# B&R Automation Studio project NAINV104C00R8L515F00 (part 10)

#### Act_OptC0011Loading.st
```iecst
ACTION Act_OptC0011Loading:
	fbLoadingWarmUpTm.PT := p_tyNtParamCurr.tComLoadRstTm ;
	udiElapseTm := (TIME_TO_UDINT (fbLoadingWarmUpTm.PT )- TIME_TO_UDINT (fbLoadingWarmUpTm.ET))/1000;
	sElapseTm := UDINT_TO_STRING(udiElapseTm);

	//Loading When Reset pressed
	IF bLoadingScreen=TRUE THEN

		fUIInRtStatOff(ADR(tyCommon.tyLoading.tyLyr.uiRtStat));
	ELSE
		fUIInRtStatHide(ADR(tyCommon.tyLoading.tyLyr.uiRtStat));
	END_IF

	IF fbLoadingWarmUpTm.Q = FALSE THEN
		tyCommon.tyLoading.tyStringMsg.sValue := CONCAT('Please wait for ',sElapseTm);
		tyCommon.tyLoading.tyStringMsg.sValue := CONCAT(tyCommon.tyLoading.tyStringMsg.sValue,' seconds...');
	END_IF

	fbLoadingWarmUpTm (IN := TRUE);
	fbLoadingLogoTm	(IN := TRUE);

	// ADD
	IF fbLoadingWarmUpTm.Q = FALSE  AND tyCommon.tyLoading.tyLyr.uiRtStat = 0 THEN
		IF fbLoadingLogoTm.Q = TRUE AND tyCommon.tyLoading.tyUILoad.usiValueIdx <= 2 THEN
			tyCommon.tyLoading.tyUILoad.usiValueIdx := (tyCommon.tyLoading.tyUILoad.usiValueIdx) +1 ;
			fbLoadingLogoTm (IN := FALSE);
			fbLoadingLogoTm (IN := TRUE);
		ELSIF fbLoadingLogoTm.Q = TRUE AND tyCommon.tyLoading.tyUILoad.usiValueIdx > 2 THEN
			tyCommon.tyLoading.tyUILoad.usiValueIdx := 0;
			fbLoadingLogoTm (IN := FALSE);
			fbLoadingLogoTm (IN := TRUE);
		END_IF
	ELSE	// fbLoadingWarmUpTm.Q = TRUE
		//fUIInRtStatHide(ADR(tyCommon.tyLoading.tyLyr.uiRtStat));
		bLoadingScreen:= FALSE;
		fbLoadingWarmUpTm (IN := FALSE);
		fbLoadingLogoTm (IN := FALSE);
	END_IF

END_ACTION
```

#### Act_EntP0000Disp.st
```iecst
ACTION Act_EntP0000Disp:

	//Access Address
	p_tyP0000SSaver ACCESS ADR(tyP0000SSaver.tySSaver);

END_ACTION
```

#### Act_OptP0000McStatus.st
```iecst
ACTION Act_OptP0000McStatus:

	IF p_bAlarmErr = TRUE THEN
		tyP0000SSaver.tySSaver.tyTxtMcStat.usiValueIdx	:= 6;

	ELSIF p_bAlarmWarning = TRUE THEN
		tyP0000SSaver.tySSaver.tyTxtMcStat.usiValueIdx	:= 7;

	ELSIF p_eOpsOpsStatus = OperationsStatusRun THEN

		tyP0000SSaver.tySSaver.tyTxtMcStat.usiValueIdx	:= 1;

//	ELSIF tyOpsProgData.bSimuCtrl = TRUE THEN
//		tyP0000SSaver.tySSaver.tyTxtMcStat.usiValueIdx	:= 5;

	ELSIF bUIManualMod = TRUE THEN
		tyP0000SSaver.tySSaver.tyTxtMcStat.usiValueIdx	:= 3;

	ELSE
		tyP0000SSaver.tySSaver.tyTxtMcStat.usiValueIdx	:= 2;

	END_IF

END_ACTION
```

#### Act_OptP0000RunningNm.st
```iecst
ACTION Act_OptP0000RunningNm:
	fbSSaverTm(IN := TRUE , PT := T#2s);

	IF EDGEPOS(fbSSaverTm.Q = FALSE) THEN
		CASE uiSSaverCnt OF
			0:
				tyP0000SSaver.tySSaver.tyTxtMcNm.sValue	:= CONCAT(p_tyMcParamCurr.sMcNm , '                                        ');
			1:
				tyP0000SSaver.tySSaver.tyTxtMcNm.sValue	:= CONCAT('          ' , CONCAT(p_tyMcParamCurr.sMcNm , '                              '));
			2:
				tyP0000SSaver.tySSaver.tyTxtMcNm.sValue	:= CONCAT('                    ' , CONCAT(p_tyMcParamCurr.sMcNm , '                    '));
			3:
				tyP0000SSaver.tySSaver.tyTxtMcNm.sValue	:= CONCAT('                              ' , CONCAT(p_tyMcParamCurr.sMcNm , '          '));
			4:
				tyP0000SSaver.tySSaver.tyTxtMcNm.sValue	:= CONCAT('                                        ' , p_tyMcParamCurr.sMcNm);
			5:
				tyP0000SSaver.tySSaver.tyTxtMcNm.sValue	:= CONCAT('                              ' , CONCAT(p_tyMcParamCurr.sMcNm , '          '));
			6:
				tyP0000SSaver.tySSaver.tyTxtMcNm.sValue	:= CONCAT('                    ' , CONCAT(p_tyMcParamCurr.sMcNm , '                    '));
			7:
				tyP0000SSaver.tySSaver.tyTxtMcNm.sValue	:= CONCAT('          ' , CONCAT(p_tyMcParamCurr.sMcNm , '                              '));

		END_CASE

	END_IF

	IF fbSSaverTm.Q = TRUE THEN
		fbSSaverTm(IN := FALSE);
		uiSSaverCnt	:= uiSSaverCnt + 1;
		IF uiSSaverCnt = 8 THEN
			uiSSaverCnt	:= 0;
		END_IF
	END_IF

END_ACTION
```

#### Act_OptP0000DisableSSaver.st
```iecst
ACTION Act_OptP0000DisableSSaver:

	IF p_tyNtParamCurr.bSSaverPrep = FALSE OR p_tyMcParamCurr.bSSaverEn = FALSE THEN

		IF tyProperty.tyVisu.uiSSaverRemainTm < 5 THEN
			tyProperty.tyVisu.uiSSaverTm	:= 9;
		ELSE
			tyProperty.tyVisu.uiSSaverTm	:= 10;
		END_IF

	END_IF

	IF EDGEPOS(p_tyNtParamCurr.bSSaverPrep AND p_tyMcParamCurr.bSSaverEn) THEN
		tyProperty.tyVisu.uiSSaverTm	:= p_tyMcParamCurr.uiSSaverTmInSec;
	END_IF

END_ACTION
```

#### Act_OptP0000StatDisp.st
```iecst
ACTION Act_OptP0000StatDisp:

	//Error / Warning / Info
	IF p_bAlarmErr = TRUE OR p_bAlarmWarning = TRUE OR p_bAlarmInfo = TRUE THEN

		fbErrBlinkTm(IN := TRUE);
		IF fbErrBlinkTm.Q = TRUE THEN
			fbErrBlinkTm(IN := FALSE);

			IF p_bAlarmErr THEN

				IF tyP0000SSaver.tySSaver.tyBitmapStat.usiValueIdx = 1 THEN
					tyP0000SSaver.tySSaver.tyBitmapStat.usiValueIdx	:= 0;
				ELSE
					tyP0000SSaver.tySSaver.tyBitmapStat.usiValueIdx	:= 1;
				END_IF

			ELSE

				IF tyP0000SSaver.tySSaver.tyBitmapStat.usiValueIdx = 3 THEN
					tyP0000SSaver.tySSaver.tyBitmapStat.usiValueIdx	:= 0;
				ELSE
					tyP0000SSaver.tySSaver.tyBitmapStat.usiValueIdx	:= 3;
				END_IF

			END_IF

		END_IF

	//Safety Relay Signal Activated
	ELSIF p_tyDI.bSafetyRlySig = FALSE THEN

		fbRstBlinkTm(IN := TRUE);
		IF fbRstBlinkTm.Q = TRUE THEN
			fbRstBlinkTm(IN := FALSE);

			IF tyP0000SSaver.tySSaver.tyBitmapStat.usiValueIdx = 5 THEN
				tyP0000SSaver.tySSaver.tyBitmapStat.usiValueIdx			:= 6;
			ELSE
				tyP0000SSaver.tySSaver.tyBitmapStat.usiValueIdx			:= 5;
			END_IF

		END_IF

	//Manual Running
	ELSIF bUIManualMod THEN
		tyP0000SSaver.tySSaver.tyBitmapStat.usiValueIdx	:= 7;

	//Operation Cycle Stopping
	ELSIF p_eOpsOpsStatus = OperationsStatusCycleStopping THEN

		fbStopBlinkTm(IN := TRUE);
		IF fbStopBlinkTm.Q = TRUE THEN
			fbStopBlinkTm(IN := FALSE);

			IF tyP0000SSaver.tySSaver.tyBitmapStat.usiValueIdx = 1 THEN
				tyP0000SSaver.tySSaver.tyBitmapStat.usiValueIdx	:= 2;
			ELSE
				tyP0000SSaver.tySSaver.tyBitmapStat.usiValueIdx	:= 1;
			END_IF

		END_IF

	//Operation Stepping
	ELSIF p_eOpsOpsStatus = OperationsStatusStep THEN
		tyP0000SSaver.tySSaver.tyBitmapStat.usiValueIdx	:= 3;

	//Operation Running
	ELSIF p_eOpsOpsStatus = OperationsStatusRun THEN
		tyP0000SSaver.tySSaver.tyBitmapStat.usiValueIdx	:= 2;

	//Standby
	ELSE
		tyP0000SSaver.tySSaver.tyBitmapStat.usiValueIdx	:= 0;

	END_IF

END_ACTION
```

#### Act_OptP0000TouchTimer.st
```iecst
ACTION Act_OptP0000TouchTimer:

	IF bLoginSuccess AND p_tyNtParamCurr.bAutoLogoutPrep AND p_tyMcParamCurr.bAutoLogoutEn THEN

		fbTouchTm();

		fbAutoLogoutTm(IN:= NOT fbTouchTm.bPressed, PT:=DINT_TO_TIME(p_tyMcParamCurr.diAutoLogoutTmInSec));

		//Reset Time When Pressed
		IF fbTouchTm.bPressed THEN
			fbAutoLogoutTm(IN:=FALSE);
		END_IF

		//Auto Logout
		IF fbAutoLogoutTm.Q THEN

			bPromptSessionExp	:= TRUE;
			p_tyC0008MsgBox ACCESS ADR(tyP0000SSaver.tyMsgBoxLoginAsk);

			IF bChgPageDone=FALSE THEN

				IF eCurrPage<>UIP0002Menu THEN
					CASE eCurrPage OF

						UIP0900GenIn, UIP0910GenOut, UIP0920MtrNPneuCtrl, UIP0923Stopper, UIP0931ConvInv, UIP0934AW, UIP0940CommCtrl:

							eChgPage		:= UIP0002Menu;

							tyP0002Menu.tyMenu.tyBtnMnlRst.bRtCompl := TRUE ;

							bChgPageDone	:= TRUE;

						UIP1000Lang, UIP1021McSetGen, UIP1022McSetVComm, UIP1023McSetHComm, UIP1024McSetAntiGap:

							IF tyCommon.tySet.tyBtnSave.uiMaskRtStat.0 = FALSE THEN

								eChgPage	:= UIP0002Menu;

								bChgPageDone	:= TRUE;

							ELSE

								eChgPage		:= UIP0002Menu;

								IF eCurrPage= UIP1021McSetGen THEN

									tyP1021McSetGen.tyMsgBoxExitAsk.tyBtnYes.bRtCompl := TRUE;

									bChgPageDone	:= TRUE;

								ELSIF eCurrPage= UIP1022McSetVComm THEN

									tyP1022McSetVComm.tyMsgBoxExitAsk.tyBtnYes.bRtCompl := TRUE;

									bChgPageDone	:= TRUE;

								ELSIF eCurrPage= UIP1023McSetHComm THEN

									tyP1023McSetHComm.tyMsgBoxExitAsk.tyBtnYes.bRtCompl := TRUE;

									bChgPageDone	:= TRUE;

								ELSIF eCurrPage= UIP1024McSetAntiGap THEN

									tyP1024McSetAntiGap.tyMsgBoxExitAsk.tyBtnYes.bRtCompl := TRUE;

									bChgPageDone	:= TRUE;

								ELSE  //language page
									bChgPageDone	:= TRUE;
								END_IF

							END_IF

						ELSE
							eChgPage		:= UIP0002Menu;

							bChgPageDone	:= TRUE;

					END_CASE

				ELSE
					bChgPageDone	:= TRUE;
				END_IF

			END_IF

			IF bChgPageDone THEN

				eUsrMgmtAct	:= UsrMgmtActLogout;

				IF p_eUsrMgmtStat = UsrMgmtActLogout AND p_eUsrMgmtStatus = Done THEN
					eUsrMgmtAct	:= UsrMgmtActIdle;

					bLoginSuccess	:= FALSE;

					bChgPageDone	:= FALSE;

					fbAutoLogoutTm(IN:=FALSE);

				END_IF

			END_IF

		END_IF

	ELSE
		fbAutoLogoutTm(IN:=FALSE);
		bChgPageDone	:= FALSE;
	END_IF

	//Prompt Relogin After Auto Logout
	IF tyP0000SSaver.tyMsgBoxLoginAsk.tyBtnYes.bRtCompl = TRUE THEN
		tyP0000SSaver.tyMsgBoxLoginAsk.tyBtnYes.bRtCompl 	:= FALSE;
		tyP0000SSaver.tyMsgBoxLoginAsk.tyBtnYes.bValue		:= FALSE;
		p_tyC0008MsgBox ACCESS ADR(tyP0000SSaver.tyMsgBoxHide);
		bPromptSessionExp	:= FALSE;

	ELSIF tyP0000SSaver.tyMsgBoxLoginAsk.tyBtnNo.bRtCompl = TRUE THEN
		tyP0000SSaver.tyMsgBoxLoginAsk.tyBtnNo.bRtCompl 	:= FALSE;
		tyP0000SSaver.tyMsgBoxLoginAsk.tyBtnNo.bValue		:= FALSE;
		p_tyC0008MsgBox ACCESS ADR(tyP0000SSaver.tyMsgBoxHide);
		eChgPage		:= UIP0100Login;
		bPromptSessionExp	:= FALSE;

	END_IF

END_ACTION
```

#### Act_EntP0001Disp.st
```iecst
ACTION Act_EntP0001Disp:

	//UI Property Access Address
	p_tyVisu ACCESS ADR(tyProperty.tyVisu);

	p_tyKeypad ACCESS ADR(tyProperty.tyKeypad);

	p_tyTxtSnippets ACCESS ADR(tyProperty.tyUITxtSnippets);

	p_tyC0008MsgBox ACCESS ADR(tyP0001Startup.tyMsgBoxHide);

	//Access Address
	p_tyP0001Startup ACCESS ADR(tyP0001Startup.tyStartup);

	p_tyP0001Initial ACCESS ADR(tyP0001Startup.tyInitial);

	fUIInRtStatHide(ADR(tyP0001Startup.tyInitial.tyLyr.uiRtStat));

END_ACTION
```

#### Act_OptP0001Startup.st
```iecst
ACTION Act_OptP0001Startup:

	//Screen Saver
	p_tyP0000SSaver ACCESS ADR(tyP0000SSaver.tySSaver);

	IF (eChgPage = UIP0001Startup) OR (eCurrPage = UIP0001Startup) THEN

		eStartupAct		:= StartupActRun;

		IF p_eStartupStat = StartupActRun AND p_eStartupStatus = Done THEN
			eStartupAct	:= StartupActIdle;

			IF p_bAlarmErr OR p_bAlarmWarning THEN
				eChgPage	:= UIP0600Alm;
			ELSE
				eChgPage	:= UIP0002Menu;
			END_IF

		END_IF

	END_IF

	tyP0001Startup.tyStartup.tyBarGraphStartup.iValue	:= DINT_TO_INT(p_eStartupStep + 1);
	tyP0001Startup.tyStartup.tyTxtStartupStat.sTxt		:= p_sStartupStepTxt;

	//IP Config
	IF DiagCpuIsSimulated() = FALSE THEN
		IF p_eStartupStep>1 THEN

			IF p_bStartupGetConfigDone THEN
				IF bTempAddrFillDone=FALSE THEN

					tyMcParamWr:= p_tyMcParamCurr;

					sTempIPAddr 	:= p_sHWInfoIPAddr;
					sTempSubnetMask	:= p_sHWInfoSubnetMask;
					udiTempEthMode	:= p_udiHWInfoEthMode;

					bTempAddrFillDone	:= TRUE;
				END_IF
			END_IF

			IF bTempAddrFillDone THEN

				IF bIPConfigChgDone=FALSE THEN

					IF  (p_tyMcParamCurr.eNetworkMod = UDINT_TO_DINT(udiTempEthMode)) AND (p_tyMcParamCurr.sIPAddr = sTempIPAddr) AND (p_tyMcParamCurr.sSubnetMask = sTempSubnetMask) THEN

						p_tyC0008MsgBox ACCESS ADR(tyP0001Startup.tyMsgBoxHide);
					ELSE
						IF p_bStartupMismatchSetConfigDone THEN

							IF (p_tyMcParamCurr.eNetworkMod <> UDINT_TO_DINT(udiTempEthMode)) THEN
								tyP0001Startup.tyMsgBoxIPConfig.tyTxtMsg.usiValueIdx := 194;
							ELSIF (p_tyMcParamCurr.sIPAddr <> sTempIPAddr) AND (p_tyMcParamCurr.sSubnetMask <> sTempSubnetMask) THEN
								tyP0001Startup.tyMsgBoxIPConfig.tyTxtMsg.usiValueIdx := 193;
							ELSIF (p_tyMcParamCurr.sIPAddr <> sTempIPAddr) THEN
								tyP0001Startup.tyMsgBoxIPConfig.tyTxtMsg.usiValueIdx := 191;
							ELSE
								tyP0001Startup.tyMsgBoxIPConfig.tyTxtMsg.usiValueIdx := 192;
							END_IF

							p_tyC0008MsgBox ACCESS ADR(tyP0001Startup.tyMsgBoxIPConfig);

						ELSE
							sSetIPAddr				:= p_tyMcParamCurr.sIPAddr;
							sSetSubnetMask			:= p_tyMcParamCurr.sSubnetMask;
							usiNetworkModeSelected	:= DINT_TO_USINT(p_tyMcParamCurr.eNetworkMod);

							bMismatchOverWriteConfig			:= TRUE;
						END_IF

					END_IF
				END_IF
			END_IF
		END_IF
	END_IF

	IF tyP0001Startup.tyMsgBoxIPConfig.tyBtnYes.bRtCompl = TRUE THEN
		tyP0001Startup.tyMsgBoxIPConfig.tyBtnYes.bRtCompl	:= FALSE;
		tyP0001Startup.tyMsgBoxIPConfig.tyBtnYes.bValue	:= FALSE;

		bIPConfigChgDone	:= TRUE;

		p_tyC0008MsgBox ACCESS ADR(tyP0001Startup.tyMsgBoxHide);

	ELSIF tyP0001Startup.tyMsgBoxIPConfig.tyBtnNo.bRtCompl = TRUE THEN

		IF (p_tyMcParamCurr.eNetworkMod <> UDINT_TO_DINT(udiTempEthMode))  THEN

			IF udiTempEthMode = DINT_TO_UDINT(IPFromDHCPServer) THEN

				bOverwriteEthMode	:= TRUE;
				bOverwriteIP 		:= FALSE;
				bOverwriteSubnet	:= FALSE;

				usiNetworkModeSelected	:= UDINT_TO_USINT(udiTempEthMode);

				tyMcParamWr.eNetworkMod	:= UDINT_TO_DINT(udiTempEthMode);

				bIPConfigChgDone	:= TRUE;

				tyP0001Startup.tyMsgBoxIPConfig.tyBtnNo.bRtCompl:= FALSE;
				tyP0001Startup.tyMsgBoxIPConfig.tyBtnNo.bValue	:= FALSE;

				p_tyC0008MsgBox ACCESS ADR(tyP0001Startup.tyMsgBoxHide);
			ELSE
				bOverwriteEthMode	:= TRUE;
				bOverwriteIP 		:= TRUE;
				bOverwriteSubnet	:= TRUE;

				usiNetworkModeSelected	:= UDINT_TO_USINT(udiTempEthMode);
				sSetIPAddr				:= sTempIPAddr;
				sSetSubnetMask			:= sTempSubnetMask;

				tyMcParamWr.eNetworkMod			:= UDINT_TO_DINT(udiTempEthMode);
				tyMcParamWr.sIPAddr				:= sTempIPAddr;
				tyMcParamWr.sSubnetMask			:= sTempSubnetMask;

				bIPConfigChgDone	:= TRUE;

				tyP0001Startup.tyMsgBoxIPConfig.tyBtnNo.bRtCompl:= FALSE;
				tyP0001Startup.tyMsgBoxIPConfig.tyBtnNo.bValue	:= FALSE;

				p_tyC0008MsgBox ACCESS ADR(tyP0001Startup.tyMsgBoxHide);
			END_IF

		ELSE

			IF (p_tyMcParamCurr.sIPAddr <> sTempIPAddr) AND (p_tyMcParamCurr.sSubnetMask <> sTempSubnetMask) THEN

				bOverwriteEthMode	:= FALSE;
				bOverwriteIP 		:= TRUE;
				bOverwriteSubnet	:= TRUE;

				sSetIPAddr		:= sTempIPAddr;
				sSetSubnetMask	:= sTempSubnetMask;

				tyMcParamWr.sIPAddr				:= sTempIPAddr;
				tyMcParamWr.sSubnetMask			:= sTempSubnetMask;

				bIPConfigChgDone	:= TRUE;

				tyP0001Startup.tyMsgBoxIPConfig.tyBtnNo.bRtCompl	:= FALSE;
				tyP0001Startup.tyMsgBoxIPConfig.tyBtnNo.bValue	:= FALSE;

				p_tyC0008MsgBox ACCESS ADR(tyP0001Startup.tyMsgBoxHide);

			ELSIF (p_tyMcParamCurr.sIPAddr <> sTempIPAddr) THEN

				bOverwriteEthMode	:= FALSE;
				bOverwriteIP 		:= TRUE;
				bOverwriteSubnet	:= FALSE;

				sSetIPAddr			:= sTempIPAddr;

				tyMcParamWr.sIPAddr	:= sTempIPAddr;

				bIPConfigChgDone	:= TRUE;

				tyP0001Startup.tyMsgBoxIPConfig.tyBtnNo.bRtCompl	:= FALSE;
				tyP0001Startup.tyMsgBoxIPConfig.tyBtnNo.bValue	:= FALSE;

				p_tyC0008MsgBox ACCESS ADR(tyP0001Startup.tyMsgBoxHide);
			ELSE

				bOverwriteEthMode	:= FALSE;
				bOverwriteIP 		:= FALSE;
				bOverwriteSubnet	:= TRUE;

				sSetSubnetMask	:= sTempSubnetMask;

				tyMcParamWr.sSubnetMask			:= sTempSubnetMask;

				bIPConfigChgDone				:= TRUE;

				tyP0001Startup.tyMsgBoxIPConfig.tyBtnNo.bRtCompl	:= FALSE;
				tyP0001Startup.tyMsgBoxIPConfig.tyBtnNo.bValue		:= FALSE;

				p_tyC0008MsgBox ACCESS ADR(tyP0001Startup.tyMsgBoxHide);
			END_IF
		END_IF
	END_IF

END_ACTION
```

#### Act_EntP0002Disp.st
```iecst
ACTION Act_EntP0002Disp:

	//Access Address
	p_tyC0005Main ACCESS ADR(tyCommon.tyMain);

	p_tyC0007Notif ACCESS ADR(tyCommon.tyNotif);

	IF NOT bPromptSessionExp THEN
		p_tyC0008MsgBox ACCESS ADR(tyP0002Menu.tyMsgBoxHide);
	END_IF

	p_tyC0009Info ACCESS ADR(tyCommon.tyInfo);

	p_tyP0002Menu ACCESS ADR(tyP0002Menu.tyMenu);

	p_tyC0011Loading ACCESS ADR(tyCommon.tyLoading);

	//Display
	//Leader Follower
	IF p_tyNtParamCurr.bLFPrep = TRUE AND p_tyMcParamCurr.bLFEn = TRUE AND ((NOT p_tyNtParamCurr.bLFUsrSetPrep AND p_tyNtParamCurr.bLeaderMc) OR (p_tyNtParamCurr.bLFUsrSetPrep AND p_tyMcParamCurr.bLFLeaderMc)) AND p_tyMcParamCurr.eUSComm <> McSetCommModHermes THEN
		fUIInRtStatOff(ADR(tyP0002Menu.tyMenu.tyBtnLFSet.uiRtStat));
		fUIInRtStatOff(ADR(tyP0002Menu.tyMenu.tyBtnLFCtrl.uiRtStat));
	ELSE
		fUIInRtStatHide(ADR(tyP0002Menu.tyMenu.tyBtnLFSet.uiRtStat));
		fUIInRtStatHide(ADR(tyP0002Menu.tyMenu.tyBtnLFCtrl.uiRtStat));
	END_IF

	//Login/Logout
	IF bLoginSuccess = FALSE THEN
		tyP0002Menu.tyMenu.tyBtnLogin.usiBitmapIdx	:= 0;
		tyP0002Menu.tyMenu.tyBtnLogin.usiTxtIdx		:= 0;
	ELSE
		tyP0002Menu.tyMenu.tyBtnLogin.usiBitmapIdx	:= 1;
		tyP0002Menu.tyMenu.tyBtnLogin.usiTxtIdx		:= 1;
	END_IF

	//Mask
	Act_OptP0002Mask;

END_ACTION
```

#### Act_OptP0002Navi.st
```iecst
ACTION Act_OptP0002Navi:

	IF (tyP0002Menu.tyMnl.tyHotspotGen.bRtCompl = TRUE) OR (tyP0002Menu.tySet.tyHotspotGen.bRtCompl = TRUE) THEN
		tyP0002Menu.tyMnl.tyHotspotGen.bRtCompl	:= FALSE;
		tyP0002Menu.tySet.tyHotspotGen.bRtCompl	:= FALSE;

		fUIInRtStatOff(ADR(tyP0002Menu.tyGen.tyLyr.uiRtStat));
		fUIInRtStatHide(ADR(tyP0002Menu.tyMnl.tyLyr.uiRtStat));
		fUIInRtStatHide(ADR(tyP0002Menu.tySet.tyLyr.uiRtStat));

	ELSIF (tyP0002Menu.tyGen.tyHotspotMnl.bRtCompl = TRUE) OR (tyP0002Menu.tySet.tyHotspotMnl.bRtCompl = TRUE) THEN
		tyP0002Menu.tyGen.tyHotspotMnl.bRtCompl	:= FALSE;
		tyP0002Menu.tySet.tyHotspotMnl.bRtCompl	:= FALSE;

		fUIInRtStatHide(ADR(tyP0002Menu.tyGen.tyLyr.uiRtStat));
		fUIInRtStatOff(ADR(tyP0002Menu.tyMnl.tyLyr.uiRtStat));
		fUIInRtStatHide(ADR(tyP0002Menu.tySet.tyLyr.uiRtStat));

	ELSIF (tyP0002Menu.tyGen.tyHotspotSet.bRtCompl = TRUE) OR (tyP0002Menu.tyMnl.tyHotspotSet.bRtCompl = TRUE) THEN
		tyP0002Menu.tyGen.tyHotspotSet.bRtCompl	:= FALSE;
		tyP0002Menu.tyMnl.tyHotspotSet.bRtCompl	:= FALSE;

		fUIInRtStatHide(ADR(tyP0002Menu.tyGen.tyLyr.uiRtStat));
		fUIInRtStatHide(ADR(tyP0002Menu.tyMnl.tyLyr.uiRtStat));
		fUIInRtStatOff(ADR(tyP0002Menu.tySet.tyLyr.uiRtStat));

	END_IF

END_ACTION
```

#### Act_OptP0002ChgPage.st
```iecst
ACTION Act_OptP0002ChgPage:

	//General
	IF tyP0002Menu.tyMenu.tyBtnOpt.bRtCompl = TRUE THEN
		tyP0002Menu.tyMenu.tyBtnOpt.bRtCompl	:= FALSE;

		eChgPage	:= UIP0200OpsGen;

	ELSIF tyP0002Menu.tyMenu.tyBtnProdSel.bRtCompl = TRUE THEN
		tyP0002Menu.tyMenu.tyBtnProdSel.bRtCompl:= FALSE;

		eChgPage	:= UIP0400ProdSel;

	ELSIF tyP0002Menu.tyMenu.tyBtnMcInfo.bRtCompl = TRUE THEN
		tyP0002Menu.tyMenu.tyBtnMcInfo.bRtCompl	:= FALSE;

		eChgPage := UIP0300McInfo;

	ELSIF tyP0002Menu.tyMenu.tyBtnAlm.bRtCompl = TRUE THEN
		tyP0002Menu.tyMenu.tyBtnAlm.bRtCompl	:= FALSE;

		eChgPage	:= UIP0600Alm;

	ELSIF tyP0002Menu.tyMenu.tyBtnLogin.bRtCompl = TRUE THEN
		tyP0002Menu.tyMenu.tyBtnLogin.bRtCompl	:= FALSE;

		eChgPage	:= UIP0100Login;

	ELSIF tyP0002Menu.tyMenu.tyBtnLFCtrl.bRtCompl = TRUE THEN
		tyP0002Menu.tyMenu.tyBtnLFCtrl.bRtCompl	:= FALSE;

		eChgPage	:= UIP0700LFCtrl;

	//Manual
	ELSIF tyP0002Menu.tyMenu.tyBtnGenInput.bRtCompl = TRUE THEN
		tyP0002Menu.tyMenu.tyBtnGenInput.bRtCompl	:= FALSE;

		bUIManualMod	:= TRUE;

		eChgPage	:= UIP0900GenIn;

	ELSIF tyP0002Menu.tyMenu.tyBtnGenOutput.bRtCompl = TRUE THEN
		tyP0002Menu.tyMenu.tyBtnGenOutput.bRtCompl	:= FALSE;

		bUIManualMod	:= TRUE;

		eChgPage	:= UIP0910GenOut;

	ELSIF tyP0002Menu.tyMenu.tyBtnMovCtrl.bRtCompl = TRUE THEN
		tyP0002Menu.tyMenu.tyBtnMovCtrl.bRtCompl	:= FALSE;

		bUIManualMod	:= TRUE;

		eChgPage	:= UIP0920MtrNPneuCtrl;

	ELSIF tyP0002Menu.tyMenu.tyBtnCommCtrl.bRtCompl = TRUE THEN
		tyP0002Menu.tyMenu.tyBtnCommCtrl.bRtCompl	:= FALSE;

		bUIManualMod	:= TRUE;

		eChgPage	:= UIP0940CommCtrl;

	ELSIF tyP0002Menu.tyMenu.tyBtnSimu.bRtCompl = TRUE THEN
		tyP0002Menu.tyMenu.tyBtnSimu.bRtCompl	:= FALSE;

		eChgPage	:= UIP0950Simu;

	//Settings
	ELSIF tyP0002Menu.tyMenu.tyBtnLang.bRtCompl = TRUE THEN
		tyP0002Menu.tyMenu.tyBtnLang.bRtCompl	:= FALSE;

		eChgPage	:= UIP1000Lang;

	ELSIF tyP0002Menu.tyMenu.tyBtnMcSet.bRtCompl = TRUE THEN
		tyP0002Menu.tyMenu.tyBtnMcSet.bRtCompl	:= FALSE;

		eChgPage	:= UIP1020McSetNavi;

	ELSIF tyP0002Menu.tyMenu.tyBtnProdSet.bRtCompl = TRUE THEN
		tyP0002Menu.tyMenu.tyBtnProdSet.bRtCompl:= FALSE;

		eChgPage	:= UIP1040ProdSet;

	ELSIF tyP0002Menu.tyMenu.tyBtnLFSet.bRtCompl = TRUE THEN
		tyP0002Menu.tyMenu.tyBtnLFSet.bRtCompl	:= FALSE;

		eChgPage	:= UIP1050LFSet;

	ELSIF tyP0002Menu.tyMenu.tyBtnUsrMgmt.bRtCompl = TRUE THEN
		tyP0002Menu.tyMenu.tyBtnUsrMgmt.bRtCompl:= FALSE;

		eChgPage	:= UIP1080UsrMgmt;

	END_IF

END_ACTION
```

#### Act_OptP0002Mask.st
```iecst
ACTION Act_OptP0002Mask:

	tyP0002Menu.tyMenu.tyBtnOpt.uiMaskRtStat.0 			:= p_tyUsrMgmtCurrAccessRgt.bOpt;
	tyP0002Menu.tyMenu.tyBtnProdSel.uiMaskRtStat.0 		:= p_tyUsrMgmtCurrAccessRgt.bProdSel AND p_bOpsStatusStop;
	tyP0002Menu.tyMenu.tyBtnMcInfo.uiMaskRtStat.0 		:= p_tyUsrMgmtCurrAccessRgt.bMcInfo;
	tyP0002Menu.tyMenu.tyBtnAlm.uiMaskRtStat.0 			:= p_tyUsrMgmtCurrAccessRgt.bAlm;
	tyP0002Menu.tyMenu.tyBtnLogin.uiMaskRtStat.0		:= p_bOpsStatusStop;
	tyP0002Menu.tyMenu.tyBtnLFCtrl.uiMaskRtStat.0 		:= p_tyUsrMgmtCurrAccessRgt.bLFCtrl;
	tyP0002Menu.tyMenu.tyBtnGenInput.uiMaskRtStat.0 	:= p_tyUsrMgmtCurrAccessRgt.bManual AND p_bOpsStatusStop;
	tyP0002Menu.tyMenu.tyBtnGenOutput.uiMaskRtStat.0 	:= p_tyUsrMgmtCurrAccessRgt.bManual AND p_bOpsStatusStop;
	tyP0002Menu.tyMenu.tyBtnMovCtrl.uiMaskRtStat.0 		:= p_tyUsrMgmtCurrAccessRgt.bManual AND p_bOpsStatusStop;
	tyP0002Menu.tyMenu.tyBtnCommCtrl.uiMaskRtStat.0 	:= p_tyUsrMgmtCurrAccessRgt.bManual AND p_bOpsStatusStop;
	tyP0002Menu.tyMenu.tyBtnSimu.uiMaskRtStat.0 		:= p_tyUsrMgmtCurrAccessRgt.bSimulation AND p_bOpsStatusStop;
	tyP0002Menu.tyMenu.tyBtnProdSet.uiMaskRtStat.0 		:= p_tyUsrMgmtCurrAccessRgt.bProdSet AND p_bOpsStatusStop;
	tyP0002Menu.tyMenu.tyBtnMcSet.uiMaskRtStat.0 		:= p_tyUsrMgmtCurrAccessRgt.bMcSet AND p_bOpsStatusStop;
	tyP0002Menu.tyMenu.tyBtnLang.uiMaskRtStat.0 		:= p_tyUsrMgmtCurrAccessRgt.bLang AND p_bOpsStatusStop;
	tyP0002Menu.tyMenu.tyBtnUsrMgmt.uiMaskRtStat.0 		:= p_tyUsrMgmtCurrAccessRgt.bUsrMgmt AND p_bOpsStatusStop;
	tyP0002Menu.tyMenu.tyBtnLFSet.uiMaskRtStat.0 		:= p_tyUsrMgmtCurrAccessRgt.bLFSet AND p_bOpsStatusStop;

	tyP0002Menu.tyMenu.tyBitmapMaskProdSetLCS.uiMaskRtStat.0	:= NOT(p_tyNtParamCurr.bLCSManageRcpPrep AND p_tyMcParamCurr.bLCSManageRcpEn);

END_ACTION
```

#### Act_OptP0002ManualCtrl.st
```iecst
ACTION Act_OptP0002ManualCtrl:

	IF EDGEPOS(bUIManualMod) THEN

		IF p_tyNtParamCurr.eTLBuzMode= TLBuzModBHTC THEN

			tyP0910GenOut.tyGenOut.tyBtnTLWhite.bValue	:= TRUE;
		ELSE

			tyP0910GenOut.tyGenOut.tyBtnTLAmber.bValue	:= TRUE;

		END_IF

		//Mask
		fUIInRtStatOff(ADR(tyP0002Menu.tyMenu.tyGenMaskLyr.uiRtStat));
		fUIInRtStatOff(ADR(tyP0002Menu.tyMenu.tySetMaskLyr.uiRtStat));

		//Show Reset Manual Button
		fUIInRtStatOff(ADR(tyP0002Menu.tyMenu.tyBtnMnlRst.uiRtStat));

	END_IF

	IF tyP0002Menu.tyMenu.tyBtnMnlRst.bRtCompl = TRUE THEN
		tyP0002Menu.tyMenu.tyBtnMnlRst.bRtCompl	:= FALSE;

		bUIManualMod	:= FALSE;

		//Unmask
		fUIInRtStatHide(ADR(tyP0002Menu.tyMenu.tyGenMaskLyr.uiRtStat));
		fUIInRtStatHide(ADR(tyP0002Menu.tyMenu.tySetMaskLyr.uiRtStat));

		//Hide Reset Manual Button
		fUIInRtStatHide(ADR(tyP0002Menu.tyMenu.tyBtnMnlRst.uiRtStat));

	END_IF

	bManualMod	:= bUIManualMod AND p_tyDI.bSafetyRlySig;

END_ACTION
```

#### Act_OptP0002UpdtData.st
```iecst
ACTION Act_OptP0002UpdtData:

	IF bLoginSuccess = FALSE THEN
		tyP0002Menu.tyMenu.tyBtnLogin.usiBitmapIdx		:= 0;
		tyP0002Menu.tyMenu.tyBtnLogin.usiTxtIdx			:= 0;
	ELSE
		tyP0002Menu.tyMenu.tyBtnLogin.usiBitmapIdx		:= 1;
		tyP0002Menu.tyMenu.tyBtnLogin.usiTxtIdx			:= 1;
	END_IF

END_ACTION
```

#### Act_OptP0002PCBReset.st
```iecst
ACTION Act_OptP0002PCBReset:

	// Product Select Hide when waiting Return Board
	IF p_bOpsInvOnceTwicePCBOut THEN

		fUIInRtStatOff(ADR(tyP0002Menu.tyMenu.tyHotspotRstRtnBrd.uiRtStat));
		fUIInRtStatHide(ADR(tyP0002Menu.tyMenu.tyBtnProdSel.uiRtStat));

		IF tyP0002Menu.tyMenu.tyHotspotRstRtnBrd.bRtCompl = TRUE THEN

			p_tyC0008MsgBox ACCESS ADR(tyP0002Menu.tyMsgBoxSelRcpWaitingBrd);

			IF tyP0002Menu.tyMsgBoxSelRcpWaitingBrd.tyBtnNo.bRtCompl = TRUE THEN
				tyP0002Menu.tyMsgBoxSelRcpWaitingBrd.tyBtnNo.bRtCompl	:= FALSE;
				tyP0002Menu.tyMsgBoxSelRcpWaitingBrd.tyBtnNo.bValue		:= FALSE;

				tyP0002Menu.tyMenu.tyHotspotRstRtnBrd.bRtCompl		 := FALSE;
				tyP0002Menu.tyMenu.tyHotspotRstRtnBrd.bValue		 := FALSE;

				p_tyC0008MsgBox ACCESS ADR(tyP0002Menu.tyMsgBoxHide);

				//Change Page
				eChgPage	:= UIP0200OpsGen;

			END_IF
		END_IF
	ELSE

		fUIInRtStatHide(ADR(tyP0002Menu.tyMenu.tyHotspotRstRtnBrd.uiRtStat));
		fUIInRtStatOff(ADR(tyP0002Menu.tyMenu.tyBtnProdSel.uiRtStat));

	END_IF

END_ACTION
```

#### Act_EntP0100Disp.st
```iecst
ACTION Act_EntP0100Disp:

	//Access Address
	p_tyC0005Main ACCESS ADR(tyCommon.tyMain);

	p_tyC0007Notif ACCESS ADR(tyCommon.tyNotif);

	p_tyC0008MsgBox ACCESS ADR(tyP0100Login.tyMsgBoxHide);

	p_tyC0009Info ACCESS ADR(tyCommon.tyInfo);

	p_tyP0100Login ACCESS ADR(tyP0100Login.tyLogin);
	p_tyP0100Logout ACCESS ADR(tyP0100Login.tyLogout);

	p_tyC0011Loading ACCESS ADR(tyCommon.tyLoading);

	//Clear Input
	tyP0100Login.tyLogin.tyStringUsrNm.sValue	:= '';
	tyP0100Login.tyLogin.tyStringPw.sValue		:= '';

	//Login Logout Layer
	IF  bLoginSuccess = TRUE THEN
		fUIInRtStatOff(ADR(tyP0100Login.tyLogout.tyLyr.uiRtStat));
		fUIInRtStatHide(ADR(tyP0100Login.tyLogin.tyLyr.uiRtStat));
	ELSE
		fUIInRtStatHide(ADR(tyP0100Login.tyLogout.tyLyr.uiRtStat));
		fUIInRtStatOff(ADR(tyP0100Login.tyLogin.tyLyr.uiRtStat));
	END_IF

	//Bypass Hotspot
	IF p_tyUsrMgmtAdminList[1].sUsrNm = '' THEN
		fUIInRtStatOff(ADR(tyP0100Login.tyLogin.tyHotspotBypassLogin.uiRtStat));
	ELSE
		fUIInRtStatHide(ADR(tyP0100Login.tyLogin.tyHotspotBypassLogin.uiRtStat));
	END_IF

	//Reset User Level Hotspot
	tyP0100Login.tyLogin.tyBtnLogin.usiBitmapIdx	:= 0;

END_ACTION
```

#### Act_OptP0100NomLogin.st
```iecst
ACTION Act_OptP0100NomLogin:

	IF tyP0100Login.tyLogin.tyBtnLogin.bRtCompl = TRUE THEN

		IF usiLoginStep = 0 THEN
			tyUsrMgmtInfoIn.sUsrNm	:= tyP0100Login.tyLogin.tyStringUsrNm.sValue;
			tyUsrMgmtInfoIn.sPw		:= tyP0100Login.tyLogin.tyStringPw.sValue;

			usiLoginStep	:= 1;

		ELSIF usiLoginStep = 1 THEN
			//User Login
			eUsrMgmtAct	:= UsrMgmtActLogin;

			IF p_eUsrMgmtStat = UsrMgmtActLogin AND p_eUsrMgmtStatus = Done THEN
				eUsrMgmtAct	:= UsrMgmtActIdle;

				IF p_bUsrMgmtNmNotExist = TRUE THEN
					usiLoginStep	:= 2;
				ELSE
					IF p_bUsrMgmtLoginSuccess = TRUE AND p_bUsrMgmtPwMismatch = FALSE THEN
						usiLoginStep	:= 3;
					ELSIF p_bUsrMgmtLoginSuccess = FALSE AND p_bUsrMgmtPwMismatch = TRUE THEN
						usiLoginStep	:= 4;
					END_IF
				END_IF

			END_IF

		ELSIF usiLoginStep = 2 THEN
			//Name Not Exist
			p_tyC0008MsgBox ACCESS ADR(tyP0100Login.tyMsgBoxNmNotExist);

			IF tyP0100Login.tyMsgBoxNmNotExist.tyBtnNo.bRtCompl = TRUE THEN
				tyP0100Login.tyMsgBoxNmNotExist.tyBtnNo.bRtCompl	:= FALSE;
				tyP0100Login.tyMsgBoxNmNotExist.tyBtnNo.bValue		:= FALSE;

				p_tyC0008MsgBox ACCESS ADR(tyP0100Login.tyMsgBoxHide);

				usiLoginStep	:= 97;
			END_IF

		ELSIF usiLoginStep = 3 THEN
			//User Login Success
			tyP1080UsrMgmt.tyUsrMgmt.tyDrpDnLvl.usiValueMinIdx 	:= 0;
			tyP1080UsrMgmt.tyUsrMgmt.tyDrpDnLvl.usiValueMaxIdx 	:= 3;

			tyP1080UsrMgmt.tyCreate.tyDrpDnLvl.usiValueMinIdx	:= 0;
			tyP1080UsrMgmt.tyCreate.tyDrpDnLvl.usiValueMaxIdx	:= 2;

			tyP1080UsrMgmt.tyEdit.tyDrpDnLvl.usiValueMinIdx		:= 0;
			tyP1080UsrMgmt.tyEdit.tyDrpDnLvl.usiValueMaxIdx		:= 2;

			usiLoginStep	:= 99;

		ELSIF usiLoginStep = 4 THEN
			//Password Mismatch
			p_tyC0008MsgBox ACCESS ADR(tyP0100Login.tyMsgBoxPwMismatch);

			IF tyP0100Login.tyMsgBoxPwMismatch.tyBtnNo.bRtCompl = TRUE THEN
				tyP0100Login.tyMsgBoxPwMismatch.tyBtnNo.bRtCompl	:= FALSE;
				tyP0100Login.tyMsgBoxPwMismatch.tyBtnNo.bValue		:= FALSE;

				p_tyC0008MsgBox ACCESS ADR(tyP0100Login.tyMsgBoxHide);

				usiLoginStep	:= 98;
			END_IF

		ELSIF usiLoginStep = 97 THEN
			tyP0100Login.tyLogin.tyStringUsrNm.sValue	:= '';
			tyP0100Login.tyLogin.tyStringPw.sValue		:= '';

			tyP0100Login.tyLogin.tyBtnLogin.bRtCompl	:= FALSE;
			tyP0100Login.tyLogin.tyBtnLogin.bValue		:= FALSE;

			usiLoginStep	:= 0;

		ELSIF usiLoginStep = 98 THEN
			//tyP0100Login.tyLogin.tyStringUsrNm.sValue	:= '';
			tyP0100Login.tyLogin.tyStringPw.sValue		:= '';

			tyP0100Login.tyLogin.tyBtnLogin.bRtCompl	:= FALSE;
			tyP0100Login.tyLogin.tyBtnLogin.bValue		:= FALSE;

			usiLoginStep	:= 0;

		ELSIF usiLoginStep = 99 THEN
			eChgPage		:= UIP0002Menu;
			bLoginSuccess	:= TRUE;

			tyP0100Login.tyLogin.tyStringUsrNm.sValue	:= '';
			tyP0100Login.tyLogin.tyStringPw.sValue		:= '';

			tyP0100Login.tyLogin.tyBtnLogin.bRtCompl	:= FALSE;
			tyP0100Login.tyLogin.tyBtnLogin.bValue		:= FALSE;

			usiLoginStep	:= 0;

		END_IF

	END_IF

END_ACTION
```

#### Act_OptP0100BypassLogin.st
```iecst
ACTION Act_OptP0100BypassLogin:

	IF tyP0100Login.tyLogin.tyHotspotBypassLogin.bRtCompl = TRUE THEN

		IF (tyP0100Login.tyLogin.tyStringUsrNm.sValue = p_tyNtParamCurr.sUIDefaultLoginNm) AND (tyP0100Login.tyLogin.tyStringPw.sValue = p_tyNtParamCurr.sUIDefaultLoginPw) THEN
			eUsrMgmtAct	:= UsrMgmtActBypassLogin;

			IF p_eUsrMgmtStat = UsrMgmtActBypassLogin AND p_eUsrMgmtStatus = Done THEN
				eUsrMgmtAct	:= UsrMgmtActIdle;

				bLoginSuccess	:= TRUE;

				//Update
				tyP1080UsrMgmt.tyUsrMgmt.tyDrpDnLvl.usiValueMinIdx	:= 0;
				tyP1080UsrMgmt.tyUsrMgmt.tyDrpDnLvl.usiValueMaxIdx	:= 3;

				tyP1080UsrMgmt.tyCreate.tyDrpDnLvl.usiValueMinIdx	:= 0;
				tyP1080UsrMgmt.tyCreate.tyDrpDnLvl.usiValueMaxIdx	:= 2;

				tyP1080UsrMgmt.tyEdit.tyDrpDnLvl.usiValueMinIdx		:= 0;
				tyP1080UsrMgmt.tyEdit.tyDrpDnLvl.usiValueMaxIdx		:= 2;

				eChgPage	:= UIP0002Menu;

				tyP0100Login.tyLogin.tyHotspotBypassLogin.bRtCompl	:= FALSE;

			END_IF

		ELSE
			p_tyC0008MsgBox ACCESS ADR(tyP0100Login.tyMsgBoxPwMismatch);

			IF tyP0100Login.tyMsgBoxPwMismatch.tyBtnNo.bRtCompl = TRUE THEN
				tyP0100Login.tyMsgBoxPwMismatch.tyBtnNo.bRtCompl	:= FALSE;
				tyP0100Login.tyMsgBoxPwMismatch.tyBtnNo.bValue		:= FALSE;

				p_tyC0008MsgBox ACCESS ADR(tyP0100Login.tyMsgBoxHide);

				tyP0100Login.tyLogin.tyStringPw.sValue		:= '';

				tyP0100Login.tyLogin.tyHotspotBypassLogin.bRtCompl	:= FALSE;

			END_IF

		END_IF

	END_IF

END_ACTION
```

#### Act_OptP0100Logout.st
```iecst
ACTION Act_OptP0100Logout:

	IF tyP0100Login.tyLogout.tyBtnLogout.bRtCompl THEN
		eUsrMgmtAct	:= UsrMgmtActLogout;

		IF p_eUsrMgmtStat = UsrMgmtActLogout AND p_eUsrMgmtStatus = Done THEN
			eUsrMgmtAct	:= UsrMgmtActIdle;

			bLoginSuccess	:= FALSE;

			//Update
			tyP0100Login.tyLogin.tyStringUsrNm.sValue		:= '';
			tyP0100Login.tyLogin.tyStringPw.sValue			:= '';

			tyP0100Login.tyLogout.tyBtnLogout.bRtCompl		:= FALSE;
			tyP0100Login.tyLogout.tyBtnLogout.bValue		:= FALSE;

			fUIInRtStatHide(ADR(tyP0100Login.tyLogout.tyLyr.uiRtStat));
			fUIInRtStatOff(ADR(tyP0100Login.tyLogin.tyLyr.uiRtStat));

		END_IF

	END_IF

END_ACTION
```

#### Act_OptP0100Keypad.st
```iecst
ACTION Act_OptP0100Keypad:

	IF fUIOutRtStatTPIsOpen(ADR(tyP0100Login.tyLogin.tyStringUsrNm.uiRtStat)) = TRUE THEN
		tyProperty.tyKeypad.tyTxtTitle.sTxt	:= tyP0100Login.tyLogin.tyStringUsrNm.sKeypadTitle;

	ELSIF fUIOutRtStatTPIsOpen(ADR(tyP0100Login.tyLogin.tyStringPw.uiRtStat)) = TRUE THEN
		tyProperty.tyKeypad.tyTxtTitle.sTxt	:= tyP0100Login.tyLogin.tyStringPw.sKeypadTitle;

	ELSE
		tyProperty.tyKeypad.tyTxtTitle.sTxt	:= '';

	END_IF

END_ACTION
```

#### Act_EntP0200Disp.st
```iecst
ACTION Act_EntP0200Disp:

	//Access Address
	p_tyC0005Main ACCESS ADR(tyCommon.tyMain);

	p_tyC0007Notif ACCESS ADR(tyCommon.tyNotif);

	p_tyC0008MsgBox ACCESS ADR(tyP0200OpsGen.tyMsgBoxHide);

	p_tyC0009Info ACCESS ADR(tyCommon.tyInfo);

	p_tyC0010RcyMsg ACCESS ADR(tyP0200OpsGen.tyRcyMsgHide);

	p_tyC0011Loading ACCESS ADR(tyCommon.tyLoading);

	p_tyP0200OpsGen ACCESS ADR(tyP0200OpsGen.tyOps);

	//Virtual Smema Layer For L to R
	p_tyP0200OpsUSVSMEMA ACCESS ADR(tyP0200OpsGen.tyUSVSMEMA);
	p_tyP0200OpsDSVSMEMA ACCESS ADR(tyP0200OpsGen.tyDSVSMEMA);

	//Virtual Smema Layer For R to L
	p_tyP0200OpsUSVSMEMA1 ACCESS ADR(tyP0200OpsGen.tyUSVSMEMA1);
	p_tyP0200OpsDSVSMEMA1 ACCESS ADR(tyP0200OpsGen.tyDSVSMEMA1);

	p_tyP0200OpsBypsInitConv ACCESS ADR(tyP0200OpsGen.tyBypsInitConv);

	//Display
	//Communication
	IF p_tyNtParamCurr.bUIConvDirRL= FALSE THEN
		IF p_tyMcParamCurr.eUSComm = McSetCommModHermes THEN
			tyP0200OpsGen.tyOps.tyBitmapUSCommIcon.usiValueIdx := 1;
		ELSIF p_tyMcParamCurr.eUSComm = McSetCommModSMEMA THEN
			tyP0200OpsGen.tyOps.tyBitmapUSCommIcon.usiValueIdx := 0;
		END_IF
		IF p_tyMcParamCurr.eDSComm = McSetCommModHermes THEN
			tyP0200OpsGen.tyOps.tyBitmapDSCommIcon.usiValueIdx := 1;
		ELSIF p_tyMcParamCurr.eDSComm = McSetCommModSMEMA THEN
			tyP0200OpsGen.tyOps.tyBitmapDSCommIcon.usiValueIdx := 0;
		END_IF
	ELSE
		IF p_tyMcParamCurr.eUSComm = McSetCommModHermes THEN
			tyP0200OpsGen.tyOps.tyBitmapDSCommIcon.usiValueIdx := 1;
		ELSIF p_tyMcParamCurr.eUSComm = McSetCommModSMEMA THEN
			tyP0200OpsGen.tyOps.tyBitmapDSCommIcon.usiValueIdx := 0;
		END_IF
		IF p_tyMcParamCurr.eDSComm = McSetCommModHermes THEN
			tyP0200OpsGen.tyOps.tyBitmapUSCommIcon.usiValueIdx := 1;
		ELSIF p_tyMcParamCurr.eDSComm = McSetCommModSMEMA THEN
			tyP0200OpsGen.tyOps.tyBitmapUSCommIcon.usiValueIdx := 0;
		END_IF
	END_IF

	//Conveyor Direction - SMEMA Arrow Indicator
	IF p_tyNtParamCurr.bUIConvDirRL THEN
		fUIInRtStatHide(ADR(tyP0200OpsGen.tyOps.tyBitmapDSCommIn.uiRtStat));
		fUIInRtStatHide(ADR(tyP0200OpsGen.tyOps.tyBitmapDSCommOut.uiRtStat));
		fUIInRtStatHide(ADR(tyP0200OpsGen.tyOps.tyBitmapUSCommIn.uiRtStat));
		fUIInRtStatHide(ADR(tyP0200OpsGen.tyOps.tyBitmapUSCommOut.uiRtStat));

		fUIInRtStatOff(ADR(tyP0200OpsGen.tyOps.tyBitmapDSCommIn1.uiRtStat));
		fUIInRtStatOff(ADR(tyP0200OpsGen.tyOps.tyBitmapDSCommOut1.uiRtStat));
		fUIInRtStatOff(ADR(tyP0200OpsGen.tyOps.tyBitmapUSCommIn1.uiRtStat));
		fUIInRtStatOff(ADR(tyP0200OpsGen.tyOps.tyBitmapUSCommOut1.uiRtStat));

		fUIInRtStatOff(ADR(tyP0200OpsGen.tyOps.tyTxtUS1.uiRtStat));
		fUIInRtStatOff(ADR(tyP0200OpsGen.tyOps.tyTxtDS1.uiRtStat));
		fUIInRtStatHide(ADR(tyP0200OpsGen.tyOps.tyTxtUS.uiRtStat));
		fUIInRtStatHide(ADR(tyP0200OpsGen.tyOps.tyTxtDS.uiRtStat));
	ELSE
		fUIInRtStatOff(ADR(tyP0200OpsGen.tyOps.tyBitmapDSCommIn.uiRtStat));
		fUIInRtStatOff(ADR(tyP0200OpsGen.tyOps.tyBitmapDSCommOut.uiRtStat));
		fUIInRtStatOff(ADR(tyP0200OpsGen.tyOps.tyBitmapUSCommIn.uiRtStat));
		fUIInRtStatOff(ADR(tyP0200OpsGen.tyOps.tyBitmapUSCommOut.uiRtStat));

		fUIInRtStatHide(ADR(tyP0200OpsGen.tyOps.tyBitmapDSCommIn1.uiRtStat));
		fUIInRtStatHide(ADR(tyP0200OpsGen.tyOps.tyBitmapDSCommOut1.uiRtStat));
		fUIInRtStatHide(ADR(tyP0200OpsGen.tyOps.tyBitmapUSCommIn1.uiRtStat));
		fUIInRtStatHide(ADR(tyP0200OpsGen.tyOps.tyBitmapUSCommOut1.uiRtStat));

		fUIInRtStatHide(ADR(tyP0200OpsGen.tyOps.tyTxtUS1.uiRtStat));
		fUIInRtStatHide(ADR(tyP0200OpsGen.tyOps.tyTxtDS1.uiRtStat));
		fUIInRtStatOff(ADR(tyP0200OpsGen.tyOps.tyTxtUS.uiRtStat));
		fUIInRtStatOff(ADR(tyP0200OpsGen.tyOps.tyTxtDS.uiRtStat));
	END_IF

	//Virtual SMEMA
	IF (p_tyUsrMgmtCurrUsr.eUsrLvl = UsrMgmtLvl1) OR p_tyNtParamCurr.bVSMEMAPrep = FALSE OR p_tyMcParamCurr.bVSMEMAEn = FALSE OR (p_tyMcParamCurr.eUSComm = McSetCommModHermes AND p_tyMcParamCurr.eDSComm = McSetCommModHermes) THEN

		tyP0200OpsGen.tyOps.tyHotspotUSVirtual.bValue	:= FALSE;
		tyP0200OpsGen.tyOps.tyHotspotDSVirtual.bValue	:= FALSE;
		tyP0200OpsGen.tyOps.tyHotspotUSVirtual1.bValue	:= FALSE;
		tyP0200OpsGen.tyOps.tyHotspotDSVirtual1.bValue	:= FALSE;

		memset(ADR(tyP0200OpsGen.tyUSVSMEMA), 0, SIZEOF(tyP0200OpsGen.tyUSVSMEMA));
		memset(ADR(tyP0200OpsGen.tyDSVSMEMA), 0, SIZEOF(tyP0200OpsGen.tyDSVSMEMA));
		memset(ADR(tyP0200OpsGen.tyUSVSMEMA1), 0, SIZEOF(tyP0200OpsGen.tyUSVSMEMA1));
		memset(ADR(tyP0200OpsGen.tyDSVSMEMA1), 0, SIZEOF(tyP0200OpsGen.tyDSVSMEMA1));

		fUIInRtStatHide(ADR(tyP0200OpsGen.tyOps.tyHotspotUSVirtual.uiRtStat));
		fUIInRtStatHide(ADR(tyP0200OpsGen.tyOps.tyHotspotDSVirtual.uiRtStat));
		fUIInRtStatHide(ADR(tyP0200OpsGen.tyUSVSMEMA.tyLyr.uiRtStat));
		fUIInRtStatHide(ADR(tyP0200OpsGen.tyDSVSMEMA.tyLyr.uiRtStat));

		fUIInRtStatHide(ADR(tyP0200OpsGen.tyOps.tyHotspotUSVirtual1.uiRtStat));
		fUIInRtStatHide(ADR(tyP0200OpsGen.tyOps.tyHotspotDSVirtual1.uiRtStat));
		fUIInRtStatHide(ADR(tyP0200OpsGen.tyUSVSMEMA1.tyLyr.uiRtStat));
		fUIInRtStatHide(ADR(tyP0200OpsGen.tyDSVSMEMA1.tyLyr.uiRtStat));

		bVSMEMAUSEn	:= FALSE;
		bVSMEMADSEn	:= FALSE;
	ELSE
		//Upstream
		IF p_tyMcParamCurr.eUSComm = McSetCommModHermes THEN
			tyP0200OpsGen.tyOps.tyHotspotUSVirtual.bValue	:= FALSE;

			memset(ADR(tyP0200OpsGen.tyUSVSMEMA), 0, SIZEOF(tyP0200OpsGen.tyUSVSMEMA));

			fUIInRtStatHide(ADR(tyP0200OpsGen.tyOps.tyHotspotUSVirtual.uiRtStat));
			fUIInRtStatHide(ADR(tyP0200OpsGen.tyUSVSMEMA.tyLyr.uiRtStat));

		ELSIF p_tyMcParamCurr.eUSComm = McSetCommModSMEMA THEN

			IF p_tyNtParamCurr.bUIConvDirRL = FALSE THEN

				tyP0200OpsGen.tyOps.tyHotspotUSVirtual.bValue	:= FALSE;

				memset(ADR(tyP0200OpsGen.tyUSVSMEMA1), 0, SIZEOF(tyP0200OpsGen.tyUSVSMEMA1));
				fUIInRtStatHide(ADR(tyP0200OpsGen.tyOps.tyHotspotUSVirtual1.uiRtStat));
				fUIInRtStatHide(ADR(tyP0200OpsGen.tyUSVSMEMA1.tyLyr.uiRtStat));

				fUIInRtStatOff(ADR(tyP0200OpsGen.tyOps.tyHotspotUSVirtual.uiRtStat));

				//Display - UBA Stat
				IF p_tyMcParamCurr.tyUSCommSMEMA.eSelection = SMEMASelIPC9851Ext THEN
					fUIInRtStatOff(ADR(tyP0200OpsGen.tyUSVSMEMA.tyBtnUBAStat.uiRtStat));
					fUIInRtStatOff(ADR(tyP0200OpsGen.tyUSVSMEMA.tyBtnDual.uiRtStat));
				ELSE
					fUIInRtStatHide(ADR(tyP0200OpsGen.tyUSVSMEMA.tyBtnUBAStat.uiRtStat));
					fUIInRtStatHide(ADR(tyP0200OpsGen.tyUSVSMEMA.tyBtnDual.uiRtStat));
				END_IF

			ELSE

				tyP0200OpsGen.tyOps.tyHotspotUSVirtual.bValue	:= FALSE;

				memset(ADR(tyP0200OpsGen.tyUSVSMEMA), 0, SIZEOF(tyP0200OpsGen.tyUSVSMEMA));
				fUIInRtStatHide(ADR(tyP0200OpsGen.tyOps.tyHotspotUSVirtual.uiRtStat));
				fUIInRtStatHide(ADR(tyP0200OpsGen.tyUSVSMEMA.tyLyr.uiRtStat));

				fUIInRtStatOff(ADR(tyP0200OpsGen.tyOps.tyHotspotUSVirtual1.uiRtStat));

				//Display - UBA Stat
				IF p_tyMcParamCurr.tyUSCommSMEMA.eSelection = SMEMASelIPC9851Ext THEN
					fUIInRtStatOff(ADR(tyP0200OpsGen.tyUSVSMEMA1.tyBtnUBAStat.uiRtStat));
					fUIInRtStatOff(ADR(tyP0200OpsGen.tyUSVSMEMA1.tyBtnDual.uiRtStat));
				ELSE
					fUIInRtStatHide(ADR(tyP0200OpsGen.tyUSVSMEMA1.tyBtnUBAStat.uiRtStat));
					fUIInRtStatHide(ADR(tyP0200OpsGen.tyUSVSMEMA1.tyBtnDual.uiRtStat));
				END_IF
			END_IF
		END_IF

		//Downstream
		IF p_tyMcParamCurr.eDSComm = McSetCommModHermes THEN
			tyP0200OpsGen.tyOps.tyHotspotDSVirtual.bValue	:= FALSE;

			memset(ADR(tyP0200OpsGen.tyDSVSMEMA), 0, SIZEOF(tyP0200OpsGen.tyDSVSMEMA));

			fUIInRtStatHide(ADR(tyP0200OpsGen.tyOps.tyHotspotDSVirtual.uiRtStat));
			fUIInRtStatHide(ADR(tyP0200OpsGen.tyDSVSMEMA.tyLyr.uiRtStat));

		ELSIF p_tyMcParamCurr.eDSComm = McSetCommModSMEMA THEN

			IF p_tyNtParamCurr.bUIConvDirRL = FALSE THEN

				tyP0200OpsGen.tyOps.tyHotspotDSVirtual1.bValue	:= FALSE;

				memset(ADR(tyP0200OpsGen.tyDSVSMEMA1), 0, SIZEOF(tyP0200OpsGen.tyDSVSMEMA1));

				fUIInRtStatHide(ADR(tyP0200OpsGen.tyOps.tyHotspotDSVirtual1.uiRtStat));
				fUIInRtStatHide(ADR(tyP0200OpsGen.tyDSVSMEMA1.tyLyr.uiRtStat));

				fUIInRtStatOff(ADR(tyP0200OpsGen.tyOps.tyHotspotDSVirtual.uiRtStat));

				//Display - DBA Stat
				IF p_tyMcParamCurr.tyDSCommSMEMA.eSelection = SMEMASelIPC9851Ext THEN
					fUIInRtStatOff(ADR(tyP0200OpsGen.tyDSVSMEMA.tyBtnDSBStat.uiRtStat));
					fUIInRtStatOff(ADR(tyP0200OpsGen.tyDSVSMEMA.tyBtnDual.uiRtStat));
				ELSE
					fUIInRtStatHide(ADR(tyP0200OpsGen.tyDSVSMEMA.tyBtnDSBStat.uiRtStat));
					fUIInRtStatHide(ADR(tyP0200OpsGen.tyDSVSMEMA.tyBtnDual.uiRtStat));
				END_IF

			ELSE

				tyP0200OpsGen.tyOps.tyHotspotDSVirtual.bValue	:= FALSE;

				memset(ADR(tyP0200OpsGen.tyDSVSMEMA), 0, SIZEOF(tyP0200OpsGen.tyDSVSMEMA));

				fUIInRtStatHide(ADR(tyP0200OpsGen.tyOps.tyHotspotDSVirtual.uiRtStat));
				fUIInRtStatHide(ADR(tyP0200OpsGen.tyDSVSMEMA.tyLyr.uiRtStat));

				fUIInRtStatOff(ADR(tyP0200OpsGen.tyOps.tyHotspotDSVirtual1.uiRtStat));

				//Display - DBA Stat
				IF p_tyMcParamCurr.tyDSCommSMEMA.eSelection = SMEMASelIPC9851Ext THEN
					fUIInRtStatOff(ADR(tyP0200OpsGen.tyDSVSMEMA1.tyBtnDSBStat.uiRtStat));
					fUIInRtStatOff(ADR(tyP0200OpsGen.tyDSVSMEMA1.tyBtnDual.uiRtStat));
				ELSE
					fUIInRtStatHide(ADR(tyP0200OpsGen.tyDSVSMEMA1.tyBtnDSBStat.uiRtStat));
					fUIInRtStatHide(ADR(tyP0200OpsGen.tyDSVSMEMA1.tyBtnDual.uiRtStat));
				END_IF

			END_IF
		END_IF

	END_IF

	//Virtual Semma Layer for Upstream2 (InvertOnce & InvertTwice_2023_0032B01)
	p_tyP0200OpsUSVSMEMA2 ACCESS ADR(tyP0200OpsGen.tyUSVSMEMA2);

	//Conveyor Direction - SMEMA Arrow Indicator (InvertOnce & InvertTwice_2023_0032B01)
	IF p_tyNtParamCurr.bProjInvertOncePrep OR p_tyNtParamCurr.bProjInvertTwicePrep THEN
		fUIInRtStatOff(ADR(tyP0200OpsGen.tyOps.tyBitmapUSCommIn2.uiRtStat));
		fUIInRtStatOff(ADR(tyP0200OpsGen.tyOps.tyBitmapUSCommOut2.uiRtStat));
	ELSE
		fUIInRtStatHide(ADR(tyP0200OpsGen.tyOps.tyBitmapUSCommIn2.uiRtStat));
		fUIInRtStatHide(ADR(tyP0200OpsGen.tyOps.tyBitmapUSCommOut2.uiRtStat));

	END_IF

	//Communication for Upstream 2 (InvertOnce & InvertTwice_2023_0032B01)
	IF p_tyNtParamCurr.bProjInvertOncePrep OR p_tyNtParamCurr.bProjInvertTwicePrep THEN
		IF p_tyMcParamCurr.eUSComm2 = McSetCommModHermes THEN
			tyP0200OpsGen.tyOps.tyBitmapUSCommIcon2.usiValueIdx	:= 1;
		ELSIF p_tyMcParamCurr.eUSComm2 = McSetCommModSMEMA THEN
			tyP0200OpsGen.tyOps.tyBitmapUSCommIcon2.usiValueIdx	:= 0;
		END_IF

	//Virtual SMEMA(InvertOnce & InvertTwice_2023_0032B01)
		IF (p_tyUsrMgmtCurrUsr.eUsrLvl = UsrMgmtLvl1) OR p_tyNtParamCurr.bVSMEMAPrep = FALSE OR p_tyMcParamCurr.bVSMEMAEn = FALSE OR (p_tyMcParamCurr.eUSComm2 = McSetCommModHermes) THEN

			tyP0200OpsGen.tyOps.tyHotspotUSVirtual2.bValue	:= FALSE;

			memset(ADR(tyP0200OpsGen.tyUSVSMEMA2), 0, SIZEOF(tyP0200OpsGen.tyUSVSMEMA2));

			fUIInRtStatHide(ADR(tyP0200OpsGen.tyOps.tyHotspotUSVirtual2.uiRtStat));
			fUIInRtStatHide(ADR(tyP0200OpsGen.tyUSVSMEMA2.tyLyr.uiRtStat));
			bVSMEMAUS2En	:= FALSE;

		ELSE
			//Upstream2
			IF p_tyMcParamCurr.eUSComm2 = McSetCommModHermes THEN
				tyP0200OpsGen.tyOps.tyHotspotUSVirtual2.bValue	:= FALSE;

				memset(ADR(tyP0200OpsGen.tyUSVSMEMA2), 0, SIZEOF(tyP0200OpsGen.tyUSVSMEMA2));

				fUIInRtStatHide(ADR(tyP0200OpsGen.tyOps.tyHotspotUSVirtual2.uiRtStat));
				fUIInRtStatHide(ADR(tyP0200OpsGen.tyUSVSMEMA2.tyLyr.uiRtStat));

			ELSIF p_tyMcParamCurr.eUSComm2 = McSetCommModSMEMA THEN

				tyP0200OpsGen.tyOps.tyHotspotUSVirtual2.bValue	:= FALSE;

				fUIInRtStatOff(ADR(tyP0200OpsGen.tyOps.tyHotspotUSVirtual2.uiRtStat));

				//Display - UBA Stat
				IF p_tyMcParamCurr.tyUSCommSMEMA2.eSelection = SMEMASelIPC9851Ext THEN
					fUIInRtStatOff(ADR(tyP0200OpsGen.tyUSVSMEMA2.tyBtnUBAStat.uiRtStat));
					fUIInRtStatOff(ADR(tyP0200OpsGen.tyUSVSMEMA2.tyBtnDual.uiRtStat));
				ELSE
					fUIInRtStatHide(ADR(tyP0200OpsGen.tyUSVSMEMA2.tyBtnUBAStat.uiRtStat));
					fUIInRtStatHide(ADR(tyP0200OpsGen.tyUSVSMEMA2.tyBtnDual.uiRtStat));
				END_IF
			END_IF
		END_IF

	END_IF

END_ACTION
```

#### Act_OptP0200ChgPage.st
```iecst
ACTION Act_OptP0200ChgPage:

	IF tyP0200OpsGen.tyOps.tyHotspotMc.bRtCompl = TRUE THEN
		tyP0200OpsGen.tyOps.tyHotspotMc.bRtCompl	:= FALSE;

		eChgPage	:= UIP0201OpsConv;
	END_IF

END_ACTION
```

#### Act_OptP0200UpdtDat.st
```iecst
ACTION Act_OptP0200UpdtDat:

	//Communication - Mask
	IF p_tyMcParamCurr.eUSComm = McSetCommModSMEMA THEN
		fUIInRtStatHide(ADR(tyP0200OpsGen.tyOps.tyBitmapUSCommIcon.uiMaskRtStat));
	ELSIF p_tyMcParamCurr.eUSComm = McSetCommModHermes THEN

		IF p_tyNtParamCurr.bUIConvDirRL= FALSE THEN
			IF p_bUSHermesConnected = TRUE THEN
				fUIInRtStatHide(ADR(tyP0200OpsGen.tyOps.tyBitmapUSCommIcon.uiMaskRtStat));
			ELSE
				fUIInRtStatOff(ADR(tyP0200OpsGen.tyOps.tyBitmapUSCommIcon.uiMaskRtStat));
			END_IF
		ELSE
			IF p_bUSHermesConnected = TRUE THEN
				fUIInRtStatHide(ADR(tyP0200OpsGen.tyOps.tyBitmapDSCommIcon.uiMaskRtStat));
			ELSE
				fUIInRtStatOff(ADR(tyP0200OpsGen.tyOps.tyBitmapDSCommIcon.uiMaskRtStat));
			END_IF
		END_IF
	END_IF

	IF p_tyMcParamCurr.eDSComm = McSetCommModSMEMA THEN
		fUIInRtStatHide(ADR(tyP0200OpsGen.tyOps.tyBitmapDSCommIcon.uiMaskRtStat));
	ELSIF p_tyMcParamCurr.eDSComm = McSetCommModHermes THEN
		IF p_tyNtParamCurr.bUIConvDirRL= FALSE THEN
			IF p_bDSHermesConnected = TRUE THEN
				fUIInRtStatHide(ADR(tyP0200OpsGen.tyOps.tyBitmapDSCommIcon.uiMaskRtStat));
			ELSE
				fUIInRtStatOff(ADR(tyP0200OpsGen.tyOps.tyBitmapDSCommIcon.uiMaskRtStat));
			END_IF
		ELSE
			IF p_bDSHermesConnected = TRUE THEN
				fUIInRtStatHide(ADR(tyP0200OpsGen.tyOps.tyBitmapUSCommIcon.uiMaskRtStat));
			ELSE
				fUIInRtStatOff(ADR(tyP0200OpsGen.tyOps.tyBitmapUSCommIcon.uiMaskRtStat));
			END_IF
		END_IF
	END_IF

	//Conv PCB Status
	IF p_bConvHvBrd = TRUE THEN
		IF p_bConvGdBrd = TRUE THEN
			tyP0200OpsGen.tyOps.tyBitmapConvPCB.usiValueIdx		:= 1;
		ELSE
			tyP0200OpsGen.tyOps.tyBitmapConvPCB.usiValueIdx		:= 2;
		END_IF
	ELSE
		tyP0200OpsGen.tyOps.tyBitmapConvPCB.usiValueIdx			:= 0;
	END_IF

	//SMEMA
	IF p_tyMcParamCurr.eUSComm = McSetCommModSMEMA THEN

		IF p_tyNtParamCurr.bUIConvDirRL = FALSE THEN
			//USB (Upstream <--- Machine)
			IF p_bUSSMEMADSRdy = TRUE THEN
				tyP0200OpsGen.tyOps.tyBitmapUSCommOut.usiValueIdx		:= 1;
			ELSE
				tyP0200OpsGen.tyOps.tyBitmapUSCommOut.usiValueIdx		:= 0;
			END_IF

			//UBA (Upstream ---> Machine)
			IF p_bUSSMEMAUSRdy = TRUE THEN
				IF p_bUSSMEMAUSGdBrdRdy = TRUE THEN
					tyP0200OpsGen.tyOps.tyBitmapUSCommIn.usiValueIdx	:= 1;
				ELSE
					tyP0200OpsGen.tyOps.tyBitmapUSCommIn.usiValueIdx	:= 2;
				END_IF
			ELSE
				tyP0200OpsGen.tyOps.tyBitmapUSCommIn.usiValueIdx		:= 0;
			END_IF
		ELSE
			// USB (Upstream <--- Machine) R TO L

			IF p_bUSSMEMADSRdy = TRUE THEN
				tyP0200OpsGen.tyOps.tyBitmapUSCommOut1.usiValueIdx		:= 1;
			ELSE
				tyP0200OpsGen.tyOps.tyBitmapUSCommOut1.usiValueIdx		:= 0;
			END_IF

			//UBA (Upstream ---> Machine) R To L
			IF p_bUSSMEMAUSRdy = TRUE THEN
				IF p_bUSSMEMAUSGdBrdRdy = TRUE THEN
					tyP0200OpsGen.tyOps.tyBitmapUSCommIn1.usiValueIdx	:= 1;
				ELSE
					tyP0200OpsGen.tyOps.tyBitmapUSCommIn1.usiValueIdx	:= 2;
				END_IF
			ELSE
				tyP0200OpsGen.tyOps.tyBitmapUSCommIn1.usiValueIdx		:= 0;
			END_IF

		END_IF

	ELSIF p_tyMcParamCurr.eUSComm = McSetCommModHermes THEN
		IF p_bUSHermesDSRdy = TRUE THEN
			IF p_bUSHermesDSGdRdy = TRUE THEN
				tyP0200OpsGen.tyOps.tyBitmapUSCommOut.usiValueIdx	:= 1;
			ELSE
				tyP0200OpsGen.tyOps.tyBitmapUSCommOut.usiValueIdx	:= 2;
			END_IF
		ELSE
			tyP0200OpsGen.tyOps.tyBitmapUSCommOut.usiValueIdx	:= 0;
		END_IF

		IF p_bUSHermesUSRdy = TRUE THEN
			IF p_bUSHermesUSGdRdy = TRUE THEN
				tyP0200OpsGen.tyOps.tyBitmapUSCommIn.usiValueIdx	:= 1;
			ELSE
				tyP0200OpsGen.tyOps.tyBitmapUSCommIn.usiValueIdx	:= 2;
			END_IF
		ELSE
			tyP0200OpsGen.tyOps.tyBitmapUSCommIn.usiValueIdx	:= 0;
		END_IF

	END_IF

	IF p_tyMcParamCurr.eDSComm = McSetCommModSMEMA THEN
		IF p_tyNtParamCurr.bUIConvDirRL = FALSE AND NOT(p_tyNtParamCurr.bProjInvertOncePrep OR p_tyNtParamCurr.bProjInvertTwicePrep) THEN
			//DBA (Machine --> Downstream)
			IF p_bDSSMEMAUSRdy = TRUE THEN
				IF p_bDSSMEMAUSGdBrdRdy = TRUE THEN
					tyP0200OpsGen.tyOps.tyBitmapDSCommOut.usiValueIdx	:= 1;
				ELSE
					tyP0200OpsGen.tyOps.tyBitmapDSCommOut.usiValueIdx	:= 2;
				END_IF
			ELSE
				tyP0200OpsGen.tyOps.tyBitmapDSCommOut.usiValueIdx		:= 0;
			END_IF

			//DSB (Machine <--- Downstream)
			IF p_bDSSMEMADSRdy = TRUE THEN
				tyP0200OpsGen.tyOps.tyBitmapDSCommIn.usiValueIdx		:= 1;
			ELSE
				tyP0200OpsGen.tyOps.tyBitmapDSCommIn.usiValueIdx		:= 0;
			END_IF

		ELSIF p_tyNtParamCurr.bProjInvertOncePrep OR p_tyNtParamCurr.bProjInvertTwicePrep THEN
			IF p_bDSSMEMAUSRdy = TRUE THEN
				tyP0200OpsGen.tyOps.tyBitmapDSCommOut.usiValueIdx	:= 1;
			ELSE
				tyP0200OpsGen.tyOps.tyBitmapDSCommOut.usiValueIdx	:= 0;
			END_IF

			//DSB (Machine <--- Downstream)
			IF p_bDSSMEMADSRdy = TRUE THEN
				tyP0200OpsGen.tyOps.tyBitmapDSCommIn.usiValueIdx		:= 1;
			ELSE
				tyP0200OpsGen.tyOps.tyBitmapDSCommIn.usiValueIdx		:= 0;
			END_IF

		ELSE

			//DBA (Machine --> Downstream) R To L
			IF p_bDSSMEMAUSRdy = TRUE THEN
				IF p_bDSSMEMAUSGdBrdRdy = TRUE THEN
					tyP0200OpsGen.tyOps.tyBitmapDSCommOut1.usiValueIdx	:= 1;
				ELSE
					tyP0200OpsGen.tyOps.tyBitmapDSCommOut1.usiValueIdx	:= 2;
				END_IF
			ELSE
				tyP0200OpsGen.tyOps.tyBitmapDSCommOut1.usiValueIdx		:= 0;
			END_IF

			//DSB (Machine <--- Downstream) R TO L
			IF p_bDSSMEMADSRdy = TRUE THEN
				tyP0200OpsGen.tyOps.tyBitmapDSCommIn1.usiValueIdx		:= 1;
			ELSE
				tyP0200OpsGen.tyOps.tyBitmapDSCommIn1.usiValueIdx		:= 0;
			END_IF

		END_IF

	ELSIF p_tyMcParamCurr.eDSComm = McSetCommModHermes THEN
		IF p_bDSHermesUSRdy = TRUE THEN
			IF p_bDSHermesUSGdRdy = TRUE THEN
				tyP0200OpsGen.tyOps.tyBitmapDSCommOut.usiValueIdx	:= 1;
			ELSE
				tyP0200OpsGen.tyOps.tyBitmapDSCommOut.usiValueIdx	:= 2;
			END_IF
		ELSE
			tyP0200OpsGen.tyOps.tyBitmapDSCommOut.usiValueIdx	:= 0;
		END_IF

		IF p_bDSHermesDSRdy = TRUE THEN
			IF p_bDSHermesDSGdRdy = TRUE THEN
				tyP0200OpsGen.tyOps.tyBitmapDSCommIn.usiValueIdx	:= 1;
			ELSE
				tyP0200OpsGen.tyOps.tyBitmapDSCommIn.usiValueIdx	:= 2;
			END_IF
		ELSE
			tyP0200OpsGen.tyOps.tyBitmapDSCommIn.usiValueIdx	:= 0;
		END_IF
	END_IF

	//Alarm
	IF NOT p_bAlarmErr THEN
		memset(ADR(tyUIAlmData.bAlm) , 0 , SIZEOF(tyUIAlmData.bAlm));
	END_IF

	IF NOT p_bAlarmWarning THEN
		memset(ADR(tyUIAlmData.bWarning) , 0 , SIZEOF(tyUIAlmData.bWarning));
	ELSE
		IF (p_bUSHermesConnected) OR p_tyMcParamCurr.eUSComm = McSetCommModSMEMA THEN
			tyUIAlmData.bWarning[3114] := FALSE;
		END_IF
		IF (p_bDSHermesConnected) OR p_tyMcParamCurr.eDSComm = McSetCommModSMEMA THEN
			tyUIAlmData.bWarning[3363] := FALSE;
		END_IF
	END_IF

	FOR i := 1 TO c_uiP0200TableSize DO
		IF p_bStartupUISettingsLoadDone THEN
			IF p_tyAlarmCurrList[i].eSeverity = AlmSeverityError THEN
				tyUIAlmData.bAlm[p_tyAlarmCurrList[i].udiErrorCode] := p_tyAlarmCurrList[i].bAlm;
			ELSIF p_tyAlarmCurrList[i].eSeverity = AlmSeverityWarning THEN
				tyUIAlmData.bWarning[p_tyAlarmCurrList[i].udiErrorCode] := p_tyAlarmCurrList[i].bWarning;
			END_IF
		END_IF
	END_FOR

	//Communication (Upstream 2) - Mask (InvertOnce & InvertTwice_2023_0032B01)
	IF p_tyMcParamCurr.eUSComm2 = McSetCommModSMEMA THEN
		fUIInRtStatHide(ADR(tyP0200OpsGen.tyOps.tyBitmapUSCommIcon2.uiMaskRtStat));
	ELSIF p_tyMcParamCurr.eUSComm2 = McSetCommModHermes THEN
		IF p_bUSHermesConnected = TRUE THEN
			fUIInRtStatHide(ADR(tyP0200OpsGen.tyOps.tyBitmapUSCommIcon2.uiMaskRtStat));
		ELSE
			fUIInRtStatOff(ADR(tyP0200OpsGen.tyOps.tyBitmapUSCommIcon2.uiMaskRtStat));
		END_IF
	END_IF
	//SMEMA (Upstream 2)(InvertOnce & InvertTwice_2023_0032B01)
	IF p_tyMcParamCurr.eUSComm2 = McSetCommModSMEMA THEN

		//USB2 (Upstream <--- Machine)
		IF p_bUSSMEMA2DSRdy = TRUE THEN
			tyP0200OpsGen.tyOps.tyBitmapUSCommOut2.usiValueIdx		:= 1;
		ELSE
			tyP0200OpsGen.tyOps.tyBitmapUSCommOut2.usiValueIdx		:= 0;
		END_IF

		//UBA2 (Upstream ---> Machine)
		IF p_bUSSMEMA2USRdy = TRUE THEN
			IF p_bUSSMEMA2USGdBrdRdy = TRUE THEN
				tyP0200OpsGen.tyOps.tyBitmapUSCommIn2.usiValueIdx	:= 1;
			ELSE
				tyP0200OpsGen.tyOps.tyBitmapUSCommIn2.usiValueIdx	:= 2;
			END_IF
		ELSE
			tyP0200OpsGen.tyOps.tyBitmapUSCommIn2.usiValueIdx		:= 0;
		END_IF

	ELSIF p_tyMcParamCurr.eUSComm2 = McSetCommModHermes THEN
		IF p_bUSHermesDSRdy = TRUE THEN
			IF p_bUSHermesDSGdRdy = TRUE THEN
				tyP0200OpsGen.tyOps.tyBitmapUSCommOut2.usiValueIdx	:= 1;
			ELSE
				tyP0200OpsGen.tyOps.tyBitmapUSCommOut2.usiValueIdx	:= 2;
			END_IF
		ELSE
			tyP0200OpsGen.tyOps.tyBitmapUSCommOut2.usiValueIdx	:= 0;
		END_IF

		IF p_bUSHermesUSRdy = TRUE THEN
			IF p_bUSHermesUSGdRdy = TRUE THEN
				tyP0200OpsGen.tyOps.tyBitmapUSCommIn2.usiValueIdx	:= 1;
			ELSE
				tyP0200OpsGen.tyOps.tyBitmapUSCommIn2.usiValueIdx	:= 2;
			END_IF
		ELSE
			tyP0200OpsGen.tyOps.tyBitmapUSCommIn2.usiValueIdx	:= 0;
		END_IF

	END_IF

END_ACTION
```

#### Act_OptP0200VSMEMA.st
```iecst
ACTION Act_OptP0200VSMEMA:

	// Virtual SMEMA - Upstream Enable/Disable
	IF p_tyNtParamCurr.bUIConvDirRL = FALSE THEN
		IF tyP0200OpsGen.tyOps.tyHotspotUSVirtual.bRtCompl = TRUE THEN
			tyP0200OpsGen.tyOps.tyHotspotUSVirtual.bRtCompl	:= FALSE;

			IF tyP0200OpsGen.tyOps.tyHotspotUSVirtual.bValue = TRUE THEN
				fUIInRtStatOff(ADR(tyP0200OpsGen.tyUSVSMEMA.tyLyr.uiRtStat));
				fUIInRtStatHide(ADR(tyP0200OpsGen.tyUSVSMEMA1.tyLyr.uiRtStat));

				bVSMEMAUSEn	:= TRUE;
			ELSE
				tyP0200OpsGen.tyUSVSMEMA.tyBtnUBA.bValue		:= FALSE;
				tyP0200OpsGen.tyUSVSMEMA.tyBtnUBAStat.bValue	:= FALSE;
				tyP0200OpsGen.tyUSVSMEMA.tyBtnDual.bValue		:= FALSE;

				bVSMEMAUSEn	:= FALSE;

				fUIInRtStatHide(ADR(tyP0200OpsGen.tyUSVSMEMA.tyLyr.uiRtStat));
				fUIInRtStatHide(ADR(tyP0200OpsGen.tyUSVSMEMA1.tyLyr.uiRtStat));
			END_IF
		END_IF
	ELSE

		IF tyP0200OpsGen.tyOps.tyHotspotUSVirtual1.bRtCompl = TRUE THEN
			tyP0200OpsGen.tyOps.tyHotspotUSVirtual1.bRtCompl	:= FALSE;

			IF tyP0200OpsGen.tyOps.tyHotspotUSVirtual1.bValue = TRUE THEN
				fUIInRtStatOff(ADR(tyP0200OpsGen.tyUSVSMEMA1.tyLyr.uiRtStat));
				fUIInRtStatHide(ADR(tyP0200OpsGen.tyUSVSMEMA.tyLyr.uiRtStat));

				bVSMEMAUSEn	:= TRUE;
			ELSE
				tyP0200OpsGen.tyUSVSMEMA1.tyBtnUBA.bValue		:= FALSE;
				tyP0200OpsGen.tyUSVSMEMA1.tyBtnUBAStat.bValue	:= FALSE;
				tyP0200OpsGen.tyUSVSMEMA1.tyBtnDual.bValue	:= FALSE;

				bVSMEMAUSEn	:= FALSE;

				fUIInRtStatHide(ADR(tyP0200OpsGen.tyUSVSMEMA.tyLyr.uiRtStat));
				fUIInRtStatHide(ADR(tyP0200OpsGen.tyUSVSMEMA1.tyLyr.uiRtStat));
			END_IF
		END_IF

	END_IF

	// Virtual SMEMA - Downstream Enable/Disable
	IF p_tyNtParamCurr.bUIConvDirRL = FALSE THEN

		IF tyP0200OpsGen.tyOps.tyHotspotDSVirtual.bRtCompl = TRUE THEN
			tyP0200OpsGen.tyOps.tyHotspotDSVirtual.bRtCompl	:= FALSE;

			IF tyP0200OpsGen.tyOps.tyHotspotDSVirtual.bValue = TRUE THEN
				fUIInRtStatOff(ADR(tyP0200OpsGen.tyDSVSMEMA.tyLyr.uiRtStat));
				fUIInRtStatHide(ADR(tyP0200OpsGen.tyDSVSMEMA1.tyLyr.uiRtStat));

				bVSMEMADSEn	:= TRUE;
			ELSE
				tyP0200OpsGen.tyDSVSMEMA.tyBtnDSB.bValue		:= FALSE;

				bVSMEMADSEn	:= FALSE;

				fUIInRtStatHide(ADR(tyP0200OpsGen.tyDSVSMEMA.tyLyr.uiRtStat));
				fUIInRtStatHide(ADR(tyP0200OpsGen.tyDSVSMEMA1.tyLyr.uiRtStat));
			END_IF
		END_IF
	ELSE

		IF tyP0200OpsGen.tyOps.tyHotspotDSVirtual1.bRtCompl = TRUE THEN
			tyP0200OpsGen.tyOps.tyHotspotDSVirtual1.bRtCompl	:= FALSE;

			IF tyP0200OpsGen.tyOps.tyHotspotDSVirtual1.bValue = TRUE THEN
				fUIInRtStatOff(ADR(tyP0200OpsGen.tyDSVSMEMA1.tyLyr.uiRtStat));
				fUIInRtStatHide(ADR(tyP0200OpsGen.tyDSVSMEMA.tyLyr.uiRtStat));

				bVSMEMADSEn	:= TRUE;
			ELSE
				tyP0200OpsGen.tyDSVSMEMA1.tyBtnDSB.bValue		:= FALSE;

				bVSMEMADSEn	:= FALSE;

				fUIInRtStatHide(ADR(tyP0200OpsGen.tyDSVSMEMA.tyLyr.uiRtStat));
				fUIInRtStatHide(ADR(tyP0200OpsGen.tyDSVSMEMA1.tyLyr.uiRtStat));
			END_IF
		END_IF

	END_IF

	// Virtual SMEMA - Upstream Control
	IF p_tyNtParamCurr.bUIConvDirRL =FALSE THEN
		IF tyP0200OpsGen.tyUSVSMEMA.tyBtnDual.bRtCompl = TRUE THEN
			tyP0200OpsGen.tyUSVSMEMA.tyBtnDual.bRtCompl	:= FALSE;

			IF tyP0200OpsGen.tyUSVSMEMA.tyBtnDual.bValue = TRUE THEN
				tyP0200OpsGen.tyUSVSMEMA.tyBtnUBA.bValue		:= TRUE;
				tyP0200OpsGen.tyUSVSMEMA.tyBtnUBAStat.bValue	:= TRUE;
			ELSE
				tyP0200OpsGen.tyUSVSMEMA.tyBtnUBA.bValue		:= FALSE;
				tyP0200OpsGen.tyUSVSMEMA.tyBtnUBAStat.bValue	:= FALSE;
			END_IF

		ELSIF tyP0200OpsGen.tyUSVSMEMA.tyBtnUBA.bRtCompl = TRUE THEN
			tyP0200OpsGen.tyUSVSMEMA.tyBtnUBA.bRtCompl	:= FALSE;

			IF tyP0200OpsGen.tyUSVSMEMA.tyBtnUBA.bValue = TRUE THEN
				IF tyP0200OpsGen.tyUSVSMEMA.tyBtnUBAStat.bValue =  TRUE THEN
					tyP0200OpsGen.tyUSVSMEMA.tyBtnDual.bValue	:= TRUE;
				END_IF
			ELSE
				tyP0200OpsGen.tyUSVSMEMA.tyBtnDual.bValue	:= FALSE;
			END_IF

		ELSIF tyP0200OpsGen.tyUSVSMEMA.tyBtnUBAStat.bRtCompl = TRUE THEN
			tyP0200OpsGen.tyUSVSMEMA.tyBtnUBAStat.bRtCompl	:= FALSE;

			IF tyP0200OpsGen.tyUSVSMEMA.tyBtnUBAStat.bValue = TRUE THEN
				IF tyP0200OpsGen.tyUSVSMEMA.tyBtnUBA.bValue =  TRUE THEN
					tyP0200OpsGen.tyUSVSMEMA.tyBtnDual.bValue	:= TRUE;
				END_IF
			ELSE
				tyP0200OpsGen.tyUSVSMEMA.tyBtnDual.bValue	:= FALSE;
			END_IF

		END_IF
	ELSE

		IF tyP0200OpsGen.tyUSVSMEMA1.tyBtnDual.bRtCompl = TRUE THEN
			tyP0200OpsGen.tyUSVSMEMA1.tyBtnDual.bRtCompl	:= FALSE;

			IF tyP0200OpsGen.tyUSVSMEMA1.tyBtnDual.bValue = TRUE THEN
				tyP0200OpsGen.tyUSVSMEMA1.tyBtnUBA.bValue		:= TRUE;
				tyP0200OpsGen.tyUSVSMEMA1.tyBtnUBAStat.bValue	:= TRUE;
			ELSE
				tyP0200OpsGen.tyUSVSMEMA1.tyBtnUBA.bValue		:= FALSE;
				tyP0200OpsGen.tyUSVSMEMA1.tyBtnUBAStat.bValue	:= FALSE;
			END_IF

		ELSIF tyP0200OpsGen.tyUSVSMEMA1.tyBtnUBA.bRtCompl = TRUE THEN
			tyP0200OpsGen.tyUSVSMEMA1.tyBtnUBA.bRtCompl	:= FALSE;

			IF tyP0200OpsGen.tyUSVSMEMA1.tyBtnUBA.bValue = TRUE THEN
				IF tyP0200OpsGen.tyUSVSMEMA1.tyBtnUBAStat.bValue =  TRUE THEN
					tyP0200OpsGen.tyUSVSMEMA1.tyBtnDual.bValue	:= TRUE;
				END_IF
			ELSE
				tyP0200OpsGen.tyUSVSMEMA1.tyBtnDual.bValue	:= FALSE;
			END_IF

		ELSIF tyP0200OpsGen.tyUSVSMEMA1.tyBtnUBAStat.bRtCompl = TRUE THEN
			tyP0200OpsGen.tyUSVSMEMA1.tyBtnUBAStat.bRtCompl	:= FALSE;

			IF tyP0200OpsGen.tyUSVSMEMA1.tyBtnUBAStat.bValue = TRUE THEN
				IF tyP0200OpsGen.tyUSVSMEMA1.tyBtnUBA.bValue =  TRUE THEN
					tyP0200OpsGen.tyUSVSMEMA1.tyBtnDual.bValue	:= TRUE;
				END_IF
			ELSE
				tyP0200OpsGen.tyUSVSMEMA1.tyBtnDual.bValue	:= FALSE;
			END_IF

		END_IF

	END_IF

	//Virtual SMEMA - Downtream Control
	IF p_tyNtParamCurr.bUIConvDirRL =FALSE THEN

		IF tyP0200OpsGen.tyDSVSMEMA.tyBtnDSB.bRtCompl = TRUE THEN
			tyP0200OpsGen.tyDSVSMEMA.tyBtnDSB.bRtCompl	:= FALSE;
		END_IF
	ELSE

		IF tyP0200OpsGen.tyDSVSMEMA1.tyBtnDSB.bRtCompl = TRUE THEN
			tyP0200OpsGen.tyDSVSMEMA1.tyBtnDSB.bRtCompl	:= FALSE;
		END_IF

	END_IF

	//Virtual SMEMA - Data
	IF p_tyNtParamCurr.bUIConvDirRL =FALSE THEN

		bVSMEMAUBA		:= tyP0200OpsGen.tyUSVSMEMA.tyBtnUBA.bValue;
		bVSMEMAUBAStat	:= tyP0200OpsGen.tyUSVSMEMA.tyBtnUBAStat.bValue;
		bVSMEMADSB		:= tyP0200OpsGen.tyDSVSMEMA.tyBtnDSB.bValue;

	ELSE

		bVSMEMAUBA		:= tyP0200OpsGen.tyUSVSMEMA1.tyBtnUBA.bValue;
		bVSMEMAUBAStat	:= tyP0200OpsGen.tyUSVSMEMA1.tyBtnUBAStat.bValue;
		bVSMEMADSB		:= tyP0200OpsGen.tyDSVSMEMA1.tyBtnDSB.bValue;

	END_IF

	// Virtual SMEMA - Upstream 2 Enable/Disable (InvertOnce & InvertTwice_2023_0032B01)
	IF tyP0200OpsGen.tyOps.tyHotspotUSVirtual2.bRtCompl = TRUE THEN
		tyP0200OpsGen.tyOps.tyHotspotUSVirtual2.bRtCompl	:= FALSE;

		IF tyP0200OpsGen.tyOps.tyHotspotUSVirtual2.bValue = TRUE THEN
			fUIInRtStatOff(ADR(tyP0200OpsGen.tyUSVSMEMA2.tyLyr.uiRtStat));
			bVSMEMAUS2En	:= TRUE;
		ELSE
			tyP0200OpsGen.tyUSVSMEMA2.tyBtnUBA.bValue		:= FALSE;
			tyP0200OpsGen.tyUSVSMEMA2.tyBtnUBAStat.bValue	:= FALSE;
			tyP0200OpsGen.tyUSVSMEMA2.tyBtnDual.bValue		:= FALSE;

			bVSMEMAUS2En	:= FALSE;

			fUIInRtStatHide(ADR(tyP0200OpsGen.tyUSVSMEMA2.tyLyr.uiRtStat));

		END_IF
	END_IF

	// Virtual SMEMA - Upstream2 Control (InvertOnce & InvertTwice_2023_0032B01)
	IF tyP0200OpsGen.tyUSVSMEMA2.tyBtnDual.bRtCompl = TRUE THEN
		tyP0200OpsGen.tyUSVSMEMA2.tyBtnDual.bRtCompl	:= FALSE;

		IF tyP0200OpsGen.tyUSVSMEMA2.tyBtnDual.bValue = TRUE THEN
			tyP0200OpsGen.tyUSVSMEMA2.tyBtnUBA.bValue		:= TRUE;
			tyP0200OpsGen.tyUSVSMEMA2.tyBtnUBAStat.bValue	:= TRUE;
		ELSE
			tyP0200OpsGen.tyUSVSMEMA2.tyBtnUBA.bValue		:= FALSE;
			tyP0200OpsGen.tyUSVSMEMA2.tyBtnUBAStat.bValue	:= FALSE;
		END_IF

	ELSIF tyP0200OpsGen.tyUSVSMEMA2.tyBtnUBA.bRtCompl = TRUE THEN
		tyP0200OpsGen.tyUSVSMEMA2.tyBtnUBA.bRtCompl	:= FALSE;

		IF tyP0200OpsGen.tyUSVSMEMA2.tyBtnUBA.bValue = TRUE THEN
			IF tyP0200OpsGen.tyUSVSMEMA2.tyBtnUBAStat.bValue =  TRUE THEN
				tyP0200OpsGen.tyUSVSMEMA2.tyBtnDual.bValue	:= TRUE;
			END_IF
		ELSE
			tyP0200OpsGen.tyUSVSMEMA2.tyBtnDual.bValue	:= FALSE;
		END_IF

	ELSIF tyP0200OpsGen.tyUSVSMEMA2.tyBtnUBAStat.bRtCompl = TRUE THEN
		tyP0200OpsGen.tyUSVSMEMA2.tyBtnUBAStat.bRtCompl	:= FALSE;

		IF tyP0200OpsGen.tyUSVSMEMA2.tyBtnUBAStat.bValue = TRUE THEN
			IF tyP0200OpsGen.tyUSVSMEMA2.tyBtnUBA.bValue =  TRUE THEN
				tyP0200OpsGen.tyUSVSMEMA2.tyBtnDual.bValue	:= TRUE;
			END_IF
		ELSE
			tyP0200OpsGen.tyUSVSMEMA2.tyBtnDual.bValue	:= FALSE;
		END_IF

	END_IF

	//Virtual SMEMA Upstream2 - Data

		bVSMEMAUBA2		:= tyP0200OpsGen.tyUSVSMEMA2.tyBtnUBA.bValue;
		bVSMEMAUBAStat2	:= tyP0200OpsGen.tyUSVSMEMA2.tyBtnUBAStat.bValue;

END_ACTION
```

#### Act_OptP0200RcyMsg.st
```iecst
ACTION Act_OptP0200RcyMsg:

	//Recovery Message
	FOR i := 1 TO c_uiP0200TableSize DO

		IF tyP0200OpsGen.tyOps.a_tyHotspotRcyMsg[i].bRtCompl = TRUE THEN
			tyP0200OpsGen.tyOps.a_tyHotspotRcyMsg[i].bRtCompl	:= FALSE;

			tyP0200OpsGen.tyRcyMsg.tyTxtMsg.udiValueIdx := p_tyAlarmRcyList[i];

			IF tyP0200OpsGen.tyRcyMsg.tyTxtMsg.udiValueIdx <> 0 THEN
				p_tyC0010RcyMsg ACCESS ADR(tyP0200OpsGen.tyRcyMsg);
			ELSE
				p_tyC0010RcyMsg ACCESS ADR(tyP0200OpsGen.tyRcyMsgHide);
			END_IF

		END_IF

	END_FOR

	// Close Recovery Message
	IF tyP0200OpsGen.tyRcyMsg.tyHotspotClose.bRtCompl = TRUE THEN
		p_tyC0010RcyMsg ACCESS ADR(tyP0200OpsGen.tyRcyMsgHide);

		tyP0200OpsGen.tyRcyMsg.tyHotspotClose.bRtCompl	:= FALSE;
	END_IF

END_ACTION
```

#### Act_OptP0200PCBReset.st
```iecst
ACTION Act_OptP0200PCBReset:

	IF p_bOpsRun THEN //Run Mode

		IF p_tyProdRcpCurrRcp1.usiMcMod = 2 OR p_tyProdRcpCurrRcp1.usiMcMod = 3 THEN
			IF p_bOpsInvOnceTwicePCBOut AND ((NOT p_bUSSMEMA2Transporting) AND (p_eConvStatus <> Busy) AND NOT(p_bLeftSen OR p_bRightSen)) THEN

				fUIInRtStatHide(ADR(tyP0200OpsGen.tyOps.tyBtnPCBReset.uiMaskRtStat));

			ELSIF p_bOpsInvOnceTwicePCBOut AND (p_bUSSMEMA2Transporting OR (p_eConvStatus = Busy) OR p_bLeftSen OR p_bRightSen OR (p_eInvertStatus = Busy) OR
				p_bConvHvBrd OR (p_eClamp1Status = Busy) OR (p_eClamp2Status = Busy) OR (p_eClamp3Status = Busy )) THEN

				fUIInRtStatOff(ADR(tyP0200OpsGen.tyOps.tyBtnPCBReset.uiMaskRtStat));

			ELSE
				fUIInRtStatOff(ADR(tyP0200OpsGen.tyOps.tyBtnPCBReset.uiMaskRtStat));
			END_IF
		ELSE
			fUIInRtStatOff(ADR(tyP0200OpsGen.tyOps.tyBtnPCBReset.uiMaskRtStat));
		END_IF

	ELSIF bManualMod OR p_bOpsStatusStop THEN // Manual Mode and Stop Mode

		IF p_bOpsInvOnceTwicePCBOut AND ((NOT p_bLeftSen) OR (NOT p_bRightSen) OR (NOT p_bConvHvBrd)) THEN
			fUIInRtStatHide(ADR(tyP0200OpsGen.tyOps.tyBtnPCBReset.uiMaskRtStat));
		ELSE
			fUIInRtStatOff(ADR(tyP0200OpsGen.tyOps.tyBtnPCBReset.uiMaskRtStat));
		END_IF

	ELSE
		fUIInRtStatOff(ADR(tyP0200OpsGen.tyOps.tyBtnPCBReset.uiMaskRtStat));
		tyP0200OpsGen.tyOps.tyBtnPCBReset.bValue := FALSE;
		bRtnBrdReset := FALSE;
	END_IF

	IF p_bOpsRun OR bManualMod OR p_bOpsStatusStop THEN
		IF 	tyP0200OpsGen.tyOps.tyBtnPCBReset.bRtCompl = TRUE THEN

			p_tyC0008MsgBox ACCESS ADR(tyP0200OpsGen.tyMsgBoxRstWaitingBrdAsk);

			IF tyP0200OpsGen.tyMsgBoxRstWaitingBrdAsk.tyBtnYes.bRtCompl = TRUE THEN
				tyP0200OpsGen.tyMsgBoxRstWaitingBrdAsk.tyBtnYes.bRtCompl	:= FALSE;
				tyP0200OpsGen.tyMsgBoxRstWaitingBrdAsk.tyBtnYes.bValue		:= FALSE;

				bRtnBrdReset := TRUE;
				p_tyC0008MsgBox ACCESS ADR(tyP0200OpsGen.tyMsgBoxHide);

				tyP0200OpsGen.tyOps.tyBtnPCBReset.bValue					:= FALSE;
				tyP0200OpsGen.tyOps.tyBtnPCBReset.bRtCompl					:= FALSE;

			ELSIF tyP0200OpsGen.tyMsgBoxRstWaitingBrdAsk.tyBtnNo.bRtCompl = TRUE THEN
				tyP0200OpsGen.tyMsgBoxRstWaitingBrdAsk.tyBtnNo.bRtCompl		:= FALSE;
				tyP0200OpsGen.tyMsgBoxRstWaitingBrdAsk.tyBtnNo.bValue		:= FALSE;
				tyP0200OpsGen.tyOps.tyBtnPCBReset.bValue					:= FALSE;
				tyP0200OpsGen.tyOps.tyBtnPCBReset.bRtCompl					:= FALSE;

				p_tyC0008MsgBox ACCESS ADR(tyP0200OpsGen.tyMsgBoxHide);

			END_IF

		END_IF

	ELSE
		p_tyC0008MsgBox ACCESS ADR(tyP0200OpsGen.tyMsgBoxHide);
	END_IF

	IF bRtnBrdReset AND p_bOpsInvOnceTwicePCBOut = FALSE AND p_bOpsInvertStepUSStandby THEN
		bRtnBrdReset := FALSE;
		tyP0200OpsGen.tyOps.tyBtnPCBReset.bValue 	:= FALSE;
		tyP0200OpsGen.tyOps.tyBtnPCBReset.bRtCompl	:= FALSE;

	ELSIF (bRtnBrdReset) AND (bManualMod OR p_bOpsStatusStop) THEN
		IF p_bOpsInvOnceTwicePCBOut = FALSE THEN
			bRtnBrdReset := FALSE;
		END_IF
	END_IF

END_ACTION
```

#### Act_EntP0201Disp.st
```iecst
ACTION Act_EntP0201Disp:

	// Access Address
	p_tyC0004Navi ACCESS ADR(tyP0201OpsConv.tyNaviBack);

	p_tyC0005Main ACCESS ADR(tyCommon.tyMain);

	p_tyC0007Notif ACCESS ADR(tyCommon.tyNotif);

	p_tyC0008MsgBox ACCESS ADR(tyP0201OpsConv.tyMsgBoxHide);

	p_tyC0009Info ACCESS ADR(tyCommon.tyInfo);

	p_tyC0011Loading ACCESS ADR(tyCommon.tyLoading);

	p_tyC0012RcpPopUp ACCESS ADR(tyP0201OpsConv.tyRcpPopUp);

	p_tyP0201OpsConv ACCESS ADR(tyP0201OpsConv.tyOps);

	p_tyP0201OpsConvIOMonitor ACCESS ADR(tyP0201OpsConv.tyIOMonitor);

	p_tyP0201OpsConvIOMonitorMacSafe ACCESS ADR(tyP0201OpsConv.tyIOMonitorXStdMachineSafety);

	p_tyP0201OpsConvIOMonitorXStd ACCESS ADR(tyP0201OpsConv.tyIOMonitorXStd);

	p_tyP0201OpsConvChgParam ACCESS ADR(tyP0201OpsConv.tyChgParam);

	p_tyP0201OpsConvBypsInitConv ACCESS ADR(tyP0201OpsConv.tyBypsInitConv);

	//Display - IO Monitor
	fUIInRtStatHide(ADR(tyP0201OpsConv.tyIOMonitor.tyLyr.uiRtStat));
	fUIInRtStatHide(ADR(tyP0201OpsConv.tyIOMonitorXStd.tyLyr.uiRtStat));
	fUIInRtStatHide(ADR(tyP0201OpsConv.tyIOMonitorXStdMachineSafety.tyLyr.uiRtStat));

	tyP0201OpsConv.tyIOMonitor.tyBtnUBAStat.uiRtStat.0		:= NOT (p_tyNtParamCurr.tyDISettings.diUBAStat > 0);
	tyP0201OpsConv.tyIOMonitor.tyBtnDBAStat.uiRtStat.0		:= NOT (p_tyNtParamCurr.tyDOSettings.diDBAStat > 0);

	tyP0201OpsConv.tyIOMonitorXStd.tyBtnUBAStat.uiRtStat.0	:= NOT (p_tyNtParamCurr.tyDISettings.diUBAStat > 0);
	tyP0201OpsConv.tyIOMonitorXStd.tyBtnDBAStat.uiRtStat.0	:= NOT (p_tyNtParamCurr.tyDOSettings.diDBAStat > 0);

	//UBA Stat
	IF p_tyMcParamCurr.tyUSCommSMEMA.bStatSigSetGd = TRUE THEN
		tyP0201OpsConv.tyIOMonitor.tyBtnUBAStat.usiTxtIdx		:= 1;
		tyP0201OpsConv.tyIOMonitorXStd.tyBtnUBAStat.usiTxtIdx	:= 1;
	ELSE
		tyP0201OpsConv.tyIOMonitor.tyBtnUBAStat.usiTxtIdx		:= 2;
		tyP0201OpsConv.tyIOMonitorXStd.tyBtnUBAStat.usiTxtIdx	:= 2;
	END_IF

	//DBA Stat
	IF p_tyMcParamCurr.tyDSCommSMEMA.bStatSigSetGd = TRUE THEN
		tyP0201OpsConv.tyIOMonitor.tyBtnDBAStat.usiTxtIdx		:= 1;
		tyP0201OpsConv.tyIOMonitorXStd.tyBtnDBAStat.usiTxtIdx	:= 1;
	ELSE
		tyP0201OpsConv.tyIOMonitor.tyBtnDBAStat.usiTxtIdx		:= 2;
		tyP0201OpsConv.tyIOMonitorXStd.tyBtnDBAStat.usiTxtIdx	:= 2;
	END_IF

	//Backup Param
	tyP0201OpsConv.tyChgParamBkUp	:= tyP0201OpsConv.tyChgParam;

END_ACTION
```

#### Act_OptP0201Navi.st
```iecst
ACTION Act_OptP0201Navi:

	IF tyP0201OpsConv.tyNaviBack.tyBtnBack.bRtCompl = TRUE THEN
		tyP0201OpsConv.tyNaviBack.tyBtnBack.bRtCompl	:= FALSE;
		tyP0201OpsConv.tyNaviBack.tyBtnBack.bValue		:= FALSE;

		eChgPage	:= UIP0200OpsGen;
	END_IF

END_ACTION
```

#### Act_OptP0201UpdtDat.st
```iecst
ACTION Act_OptP0201UpdtDat:

	//Machine Status
	fbMcStatUpdtTm(IN := TRUE);
	IF fbMcStatUpdtTm.Q = TRUE THEN
		fbMcStatUpdtTm(IN := FALSE);

		IF p_bOpsUSStandby = TRUE THEN
			IF p_tyNtParamCurr.bUSWidthChkPrep AND p_tyMcParamCurr.bUSWidthChkEn AND p_tyDI.bUSWidthChkSen=FALSE THEN
				tyP0201OpsConv.tyOps.tyStringMcStatus.sValue	:= 'Width Check Sensor Block Upstream';
			ELSIF p_tyNtParamCurr.bLFPrep AND p_tyMcParamCurr.bLFEn AND p_bLFFollowerUSAllow=FALSE THEN
				tyP0201OpsConv.tyOps.tyStringMcStatus.sValue	:= 'Leader Issue Block Upstream';
			ELSE
				tyP0201OpsConv.tyOps.tyStringMcStatus.sValue	:= p_sOpsInvertStepTxt;
			END_IF
		ELSIF p_bOpsDSStandby = TRUE THEN
			IF p_tyNtParamCurr.bDSWidthChkPrep AND p_tyMcParamCurr.bDSWidthChkEn AND p_tyDI.bDSWidthChkSen=FALSE THEN
				tyP0201OpsConv.tyOps.tyStringMcStatus.sValue	:= 'Width Check Sensor Block Downstream';
			ELSIF p_tyNtParamCurr.bLFPrep AND p_tyMcParamCurr.bLFEn AND p_bLFFollowerDSAllow=FALSE THEN
				tyP0201OpsConv.tyOps.tyStringMcStatus.sValue	:= 'Leader Issue Block Downstream';
			ELSE
				tyP0201OpsConv.tyOps.tyStringMcStatus.sValue	:= p_sOpsInvertStepTxt;
			END_IF
		ELSE
			tyP0201OpsConv.tyOps.tyStringMcStatus.sValue	:= p_sOpsInvertStepTxt;
		END_IF

	END_IF

	//Mode
	tyP0201OpsConv.tyOps.tyTxtMod.usiValueIdx	:= p_tyProdRcpCurrRcp1.usiMcMod;

	//Width
	IF p_tyNtParamCurr.bAWPrep = FALSE OR p_tyMcParamCurr.bAWDis = TRUE THEN
		tyP0201OpsConv.tyOps.tyNumProdWidth.diValue	:= p_tyProdRcpCurrRcp1.diWidthInUM;
	ELSE
		tyP0201OpsConv.tyOps.tyNumProdWidth.diValue	:= p_tyMcParamCurr.diWidthAtHmPosInUM - p_diAWOpenActualPos;
	END_IF

	//Program Info
	tyP0201OpsConv.tyOps.tyStringProdNm.sValue			:= p_tyProdRcpCurrRcp1.sRcpNm;
	tyP0201OpsConv.tyOps.tyTxtFlippedBrd.usiValueIdx	:= p_tyProdRcpCurrRcp1.usiFlippedBrd;
	tyP0201OpsConv.tyOps.tyStringMatchCode.sValue		:= p_tyProdRcpCurrRcp1.sMatchCode;

	//Conveyor PCB Status
	IF p_bConvHvBrd = TRUE THEN
		IF p_bConvGdBrd = TRUE THEN
			tyP0201OpsConv.tyOps.tyBitmapConvPCB.usiValueIdx	:= 1;
		ELSE
			tyP0201OpsConv.tyOps.tyBitmapConvPCB.usiValueIdx	:= 2;
		END_IF
	ELSE
		tyP0201OpsConv.tyOps.tyBitmapConvPCB.usiValueIdx	:= 0;
	END_IF

	IF p_tyNtParamCurr.bHermesPrep=TRUE THEN
		IF p_tyMcParamCurr.eUSComm = McSetCommModSMEMA AND p_tyMcParamCurr.eDSComm = McSetCommModSMEMA THEN
			fUIInRtStatHide(ADR(tyP0201OpsConv.tyOps.tyTxtFlippedBrd.uiRtStat));
			fUIInRtStatHide(ADR(tyP0201OpsConv.tyOps.tyLblFlippedBrd.uiRtStat));
		ELSE
			fUIInRtStatOff(ADR(tyP0201OpsConv.tyOps.tyTxtFlippedBrd.uiRtStat));
			fUIInRtStatOff(ADR(tyP0201OpsConv.tyOps.tyLblFlippedBrd.uiRtStat));
		END_IF
	ELSE
		fUIInRtStatHide(ADR(tyP0201OpsConv.tyOps.tyTxtFlippedBrd.uiRtStat));
		fUIInRtStatHide(ADR(tyP0201OpsConv.tyOps.tyLblFlippedBrd.uiRtStat));
	END_IF

	//Product Recipe 254
	tyP0201OpsConv.tyOps.tyHotspotShowLRcp.uiRtStat.0 := NOT(tyP0201OpsConv.tyOps.tyStringProdNm.sValue <> '');

	IF tyP0201OpsConv.tyOps.tyHotspotShowLRcp.bRtCompl = TRUE THEN
		tyP0201OpsConv.tyOps.tyHotspotShowLRcp.bRtCompl := FALSE;

		fUIInRtStatOff(ADR(tyP0201OpsConv.tyRcpPopUp.tyLyr.uiRtStat));

		tyP0201OpsConv.tyRcpPopUp.tyStringInfo.sValue  := p_tyProdRcpCurrRcp1.sRcpNm;

	ELSIF tyP0201OpsConv.tyRcpPopUp.tyHotspotClose.bRtCompl = TRUE THEN
		tyP0201OpsConv.tyRcpPopUp.tyHotspotClose.bRtCompl := FALSE;

		fUIInRtStatHide(ADR(tyP0201OpsConv.tyRcpPopUp.tyLyr.uiRtStat));

	END_IF

END_ACTION
```

#### Act_OptP0201IOMonitor.st
```iecst
ACTION Act_OptP0201IOMonitor:

	IF tyP0201OpsConv.tyOps.tyHotspotIOMonitor.bRtCompl = TRUE THEN
		tyP0201OpsConv.tyOps.tyHotspotIOMonitor.bRtCompl	:= FALSE;

		IF ((p_tyNtParamCurr.bProjClampPrep=FALSE) OR (p_tyNtParamCurr.bProjClampPrep=TRUE AND p_tyNtParamCurr.eProjClampOption=ClampNoRS))THEN
			fUIInRtStatOff(ADR(tyP0201OpsConv.tyIOMonitor.tyLyr.uiRtStat));
			fUIInRtStatHide(ADR(tyP0201OpsConv.tyIOMonitorXStd.tyLyr.uiRtStat));
			fUIInRtStatHide(ADR(tyP0201OpsConv.tyIOMonitorXStdMachineSafety.tyLyr.uiRtStat));
		ELSIF (p_tyNtParamCurr.bProjClampPrep=TRUE) AND (p_tyNtParamCurr.bUnlockCoverPrep OR p_tyNtParamCurr.bUSDSMachineSafetySig) THEN
			fUIInRtStatHide(ADR(tyP0201OpsConv.tyIOMonitor.tyLyr.uiRtStat));
			fUIInRtStatHide(ADR(tyP0201OpsConv.tyIOMonitorXStd.tyLyr.uiRtStat));
			fUIInRtStatOff(ADR(tyP0201OpsConv.tyIOMonitorXStdMachineSafety.tyLyr.uiRtStat));
		ELSE
			fUIInRtStatHide(ADR(tyP0201OpsConv.tyIOMonitor.tyLyr.uiRtStat));
			fUIInRtStatOff(ADR(tyP0201OpsConv.tyIOMonitorXStd.tyLyr.uiRtStat));
			fUIInRtStatHide(ADR(tyP0201OpsConv.tyIOMonitorXStdMachineSafety.tyLyr.uiRtStat));
		END_IF

		// ADD increase when bProjClamp Prep and Machine Safety Signal

		p_tyC0004Navi ACCESS ADR(tyP0201OpsConv.tyNaviHide);

	ELSIF tyP0201OpsConv.tyIOMonitor.tyHotspotClose.bRtCompl = TRUE THEN
		tyP0201OpsConv.tyIOMonitor.tyHotspotClose.bRtCompl	:= FALSE;

		fUIInRtStatHide(ADR(tyP0201OpsConv.tyIOMonitor.tyLyr.uiRtStat));

		p_tyC0004Navi ACCESS ADR(tyP0201OpsConv.tyNaviBack);

	ELSIF tyP0201OpsConv.tyIOMonitorXStd.tyHotspotClose.bRtCompl = TRUE THEN
		tyP0201OpsConv.tyIOMonitorXStd.tyHotspotClose.bRtCompl	:= FALSE;

		fUIInRtStatHide(ADR(tyP0201OpsConv.tyIOMonitorXStd.tyLyr.uiRtStat));

		p_tyC0004Navi ACCESS ADR(tyP0201OpsConv.tyNaviBack);
	ELSIF tyP0201OpsConv.tyIOMonitorXStdMachineSafety.tyHotspotClose.bRtCompl = TRUE THEN
		tyP0201OpsConv.tyIOMonitorXStdMachineSafety.tyHotspotClose.bRtCompl	:= FALSE;

		fUIInRtStatHide(ADR(tyP0201OpsConv.tyIOMonitorXStdMachineSafety.tyLyr.uiRtStat));

		p_tyC0004Navi ACCESS ADR(tyP0201OpsConv.tyNaviBack);
	END_IF

	IF tyP0201OpsConv.tyIOMonitor.tyLyr.uiRtStat.0 = FALSE THEN
		//Standard
		//Digital Input
		tyP0201OpsConv.tyIOMonitor.tyBtnSafetyRlySig.bValue					:= p_tyDI.bSafetyRlySig;
		tyP0201OpsConv.tyIOMonitor.tyBtnEStop.bValue						:= p_tyDI.bEStopSig;
		tyP0201OpsConv.tyIOMonitor.tyBtnCoverSWSig.bValue					:= p_tyDI.bCoverSWSig;
		tyP0201OpsConv.tyIOMonitor.tyBtnUBA.bValue							:= p_tyDI.bUBA;
		tyP0201OpsConv.tyIOMonitor.tyBtnDSB.bValue							:= p_tyDI.bDSB;
		tyP0201OpsConv.tyIOMonitor.tyBtnUBAStat.bValue						:= p_tyDI.bUBAStat;
		tyP0201OpsConv.tyIOMonitor.tyBtnConvLftSen.bValue					:= p_tyDI.bConvLftSen;
		tyP0201OpsConv.tyIOMonitor.tyBtnConvRgtSen.bValue					:= p_tyDI.bConvRgtSen;
		tyP0201OpsConv.tyIOMonitor.tyBtnPressureSW.bValue					:= p_tyDI.bPressureSW;
		tyP0201OpsConv.tyIOMonitor.tyBtnThermalPrtSig.bValue				:= p_tyDI.bThermalPrtSig;
		tyP0201OpsConv.tyIOMonitor.tyBtnCoatingSen.bValue					:= p_tyDI.bCoatingSen;
		tyP0201OpsConv.tyIOMonitor.tyBtnUSWidthChkSen.bValue				:= p_tyDI.bUSWidthChkSen;
		tyP0201OpsConv.tyIOMonitor.tyBtnDSWidthChkSen.bValue				:= p_tyDI.bDSWidthChkSen;
		tyP0201OpsConv.tyIOMonitor.tyBtnInvertHomeSen.bValue				:= p_tyDI.bInvertHomeSen;
		tyP0201OpsConv.tyIOMonitor.tyBtnInvertRemoteSen.bValue				:= p_tyDI.bInvertRemoteSen;
		tyP0201OpsConv.tyIOMonitor.tyBtnInletShutterOpenRS.bValue			:= p_tyDI.bInShutterOpenRS;
		tyP0201OpsConv.tyIOMonitor.tyBtnInletShutterCloseRS.bValue			:= p_tyDI.bInShutterCloseRS;
		tyP0201OpsConv.tyIOMonitor.tyBtnOutletShutterOpenRS.bValue			:= p_tyDI.bOutShutterOpenRS;
		tyP0201OpsConv.tyIOMonitor.tyBtnOutletShutterCloseRS.bValue			:= p_tyDI.bOutShutterCloseRS;

		//Digital Output
		tyP0201OpsConv.tyIOMonitor.tyBtnSafetyRlyRst.bValue					:= p_tyDO.bSafetyRlyRst;
		tyP0201OpsConv.tyIOMonitor.tyBtnTLGreen.bValue						:= p_tyDO.bTLGreen;
		tyP0201OpsConv.tyIOMonitor.tyBtnTLAmber.bValue						:= p_tyDO.bTLAmber;
		tyP0201OpsConv.tyIOMonitor.tyBtnTLRed.bValue						:= p_tyDO.bTLRed;
		tyP0201OpsConv.tyIOMonitor.tyBtnTLBlue.bValue						:= p_tyDO.bTLBlue;
		tyP0201OpsConv.tyIOMonitor.tyBtnTLWhite.bValue						:= p_tyDO.bTLWhite;
		tyP0201OpsConv.tyIOMonitor.tyBtnBuzzer.bValue						:= p_tyDO.bBuz;
		tyP0201OpsConv.tyIOMonitor.tyBtnCoatingRetCtrl.bValue				:= p_tyDO.bCoatingStprRet;
		tyP0201OpsConv.tyIOMonitor.tyBtnUSB.bValue							:= p_tyDO.bUSB;
		tyP0201OpsConv.tyIOMonitor.tyBtnDBA.bValue							:= p_tyDO.bDBA;
		tyP0201OpsConv.tyIOMonitor.tyBtnDBAStat.bValue						:= p_tyDO.bDBAStat;
		tyP0201OpsConv.tyIOMonitor.tyBtnConvMtrCW.bValue					:= p_tyDO.bConvMtrCW;
		tyP0201OpsConv.tyIOMonitor.tyBtnConvMtrCCW.bValue					:= p_tyDO.bConvMtrCCW;
		tyP0201OpsConv.tyIOMonitor.tyBtnStprUnblkCtrl.bValue				:= p_tyDO.bStprUnblkCtrl;
		tyP0201OpsConv.tyIOMonitor.tyBtnStprBlkCtrl.bValue					:= p_tyDO.bStprBlkCtrl;
		tyP0201OpsConv.tyIOMonitor.tyBtnInvertHome.bValue					:= p_tyDO.bInvertHome;
		tyP0201OpsConv.tyIOMonitor.tyBtnInvertRemote.bValue					:= p_tyDO.bInvertRemote;
		tyP0201OpsConv.tyIOMonitor.tyBtnInvertBrake.bValue					:= p_tyDO.bInvertBrake;
		tyP0201OpsConv.tyIOMonitor.tyBtnClampCtrl.bValue					:= p_tyDO.bClampControl;
		tyP0201OpsConv.tyIOMonitor.tyBtnUnclampCtrl.bValue					:= p_tyDO.bUnclampControl;
		tyP0201OpsConv.tyIOMonitor.tyBtnMtrPwrRly.bValue					:= p_tyDO.bMtrPwrRly;
		tyP0201OpsConv.tyIOMonitor.tyBtnInShutterOpenCtrl.bValue			:= p_tyDO.bInShutterOpenCtrl;
		tyP0201OpsConv.tyIOMonitor.tyBtnInShutterCloseCtrl.bValue			:= p_tyDO.bInShutterCloseCtrl;
		tyP0201OpsConv.tyIOMonitor.tyBtnOutShutterOpenCtrl.bValue			:= p_tyDO.bOutShutterOpenCtrl;
		tyP0201OpsConv.tyIOMonitor.tyBtnOutShutterCloseCtrl.bValue			:= p_tyDO.bOutShutterCloseCtrl;

	END_IF

	IF tyP0201OpsConv.tyIOMonitorXStd.tyLyr.uiRtStat.0 = FALSE THEN
		//Non Standard
		//Digital Input
		tyP0201OpsConv.tyIOMonitorXStd.tyBtnSafetyRlySig.bValue					:= p_tyDI.bSafetyRlySig;
		tyP0201OpsConv.tyIOMonitorXStd.tyBtnEStop.bValue						:= p_tyDI.bEStopSig;
		tyP0201OpsConv.tyIOMonitorXStd.tyBtnCoverSWSig.bValue					:= p_tyDI.bCoverSWSig;
		tyP0201OpsConv.tyIOMonitorXStd.tyBtnUBA.bValue							:= p_tyDI.bUBA;
		tyP0201OpsConv.tyIOMonitorXStd.tyBtnDSB.bValue							:= p_tyDI.bDSB;
		tyP0201OpsConv.tyIOMonitorXStd.tyBtnUBAStat.bValue						:= p_tyDI.bUBAStat;
		tyP0201OpsConv.tyIOMonitorXStd.tyBtnUBA2.bValue							:= p_tyDI.bUBA2;
		tyP0201OpsConv.tyIOMonitorXStd.tyBtnUBAStat2.bValue						:= p_tyDI.bUBAStat2;
		tyP0201OpsConv.tyIOMonitorXStd.tyBtnConvLftSen.bValue					:= p_tyDI.bConvLftSen;
		tyP0201OpsConv.tyIOMonitorXStd.tyBtnConvRgtSen.bValue					:= p_tyDI.bConvRgtSen;
		tyP0201OpsConv.tyIOMonitorXStd.tyBtnPressureSW.bValue					:= p_tyDI.bPressureSW;
		tyP0201OpsConv.tyIOMonitorXStd.tyBtnThermalPrtSig.bValue				:= p_tyDI.bThermalPrtSig;
		tyP0201OpsConv.tyIOMonitorXStd.tyBtnCoatingSen.bValue					:= p_tyDI.bCoatingSen;
		tyP0201OpsConv.tyIOMonitorXStd.tyBtnUSWidthChkSen.bValue				:= p_tyDI.bUSWidthChkSen;
		tyP0201OpsConv.tyIOMonitorXStd.tyBtnDSWidthChkSen.bValue				:= p_tyDI.bDSWidthChkSen;
		tyP0201OpsConv.tyIOMonitorXStd.tyBtnInvertHomeSen.bValue				:= p_tyDI.bInvertHomeSen;
		tyP0201OpsConv.tyIOMonitorXStd.tyBtnInvertRemoteSen.bValue				:= p_tyDI.bInvertRemoteSen;
		tyP0201OpsConv.tyIOMonitorXStd.tyBtnInletShutterOpenRS.bValue			:= p_tyDI.bInShutterOpenRS;
		tyP0201OpsConv.tyIOMonitorXStd.tyBtnInletShutterCloseRS.bValue			:= p_tyDI.bInShutterCloseRS;
		tyP0201OpsConv.tyIOMonitorXStd.tyBtnOutletShutterOpenRS.bValue			:= p_tyDI.bOutShutterOpenRS;
		tyP0201OpsConv.tyIOMonitorXStd.tyBtnOutletShutterCloseRS.bValue			:= p_tyDI.bOutShutterCloseRS;
		tyP0201OpsConv.tyIOMonitorXStd.tyBtnClamp2Sen.bValue					:= p_tyDI.bClamp2Sen;
		tyP0201OpsConv.tyIOMonitorXStd.tyBtnClamp3Sen.bValue					:= p_tyDI.bClamp3Sen;
		tyP0201OpsConv.tyIOMonitorXStd.tyBtnClampRS1.bValue						:= p_tyDI.bClampRS1;
		tyP0201OpsConv.tyIOMonitorXStd.tyBtnUnClampRS1.bValue					:= p_tyDI.bUnClampRS1;
		tyP0201OpsConv.tyIOMonitorXStd.tyBtnClampRS2.bValue						:= p_tyDI.bClampRS2;
		tyP0201OpsConv.tyIOMonitorXStd.tyBtnUnClampRS2.bValue					:= p_tyDI.bUnClampRS2;
		tyP0201OpsConv.tyIOMonitorXStd.tyBtnClampRS3.bValue						:= p_tyDI.bClampRS3;
		tyP0201OpsConv.tyIOMonitorXStd.tyBtnUnClampRS3.bValue					:= p_tyDI.bUnClampRS3;

		//Digital Output
		tyP0201OpsConv.tyIOMonitorXStd.tyBtnSafetyRlyRst.bValue					:= p_tyDO.bSafetyRlyRst;
		tyP0201OpsConv.tyIOMonitorXStd.tyBtnTLGreen.bValue						:= p_tyDO.bTLGreen;
		tyP0201OpsConv.tyIOMonitorXStd.tyBtnTLAmber.bValue						:= p_tyDO.bTLAmber;
		tyP0201OpsConv.tyIOMonitorXStd.tyBtnTLRed.bValue						:= p_tyDO.bTLRed;
		tyP0201OpsConv.tyIOMonitorXStd.tyBtnTLBlue.bValue						:= p_tyDO.bTLBlue;
		tyP0201OpsConv.tyIOMonitorXStd.tyBtnTLWhite.bValue						:= p_tyDO.bTLWhite;
		tyP0201OpsConv.tyIOMonitorXStd.tyBtnBuzzer.bValue						:= p_tyDO.bBuz;
		tyP0201OpsConv.tyIOMonitorXStd.tyBtnCoatingRetCtrl.bValue				:= p_tyDO.bCoatingStprRet;
		tyP0201OpsConv.tyIOMonitorXStd.tyBtnUSB.bValue							:= p_tyDO.bUSB;
		tyP0201OpsConv.tyIOMonitorXStd.tyBtnDBA.bValue							:= p_tyDO.bDBA;
		tyP0201OpsConv.tyIOMonitorXStd.tyBtnDBAStat.bValue						:= p_tyDO.bDBAStat;
		tyP0201OpsConv.tyIOMonitorXStd.tyBtnUSB2.bValue							:= p_tyDO.bUSB2;
		tyP0201OpsConv.tyIOMonitorXStd.tyBtnConvMtrCW.bValue					:= p_tyDO.bConvMtrCW;
		tyP0201OpsConv.tyIOMonitorXStd.tyBtnConvMtrCCW.bValue					:= p_tyDO.bConvMtrCCW;
		tyP0201OpsConv.tyIOMonitorXStd.tyBtnInvertHome.bValue					:= p_tyDO.bInvertHome;
		tyP0201OpsConv.tyIOMonitorXStd.tyBtnInvertRemote.bValue					:= p_tyDO.bInvertRemote;
		tyP0201OpsConv.tyIOMonitorXStd.tyBtnInvertBrake.bValue					:= p_tyDO.bInvertBrake;
		tyP0201OpsConv.tyIOMonitorXStd.tyBtnMtrPwrRly.bValue					:= p_tyDO.bMtrPwrRly;
		tyP0201OpsConv.tyIOMonitorXStd.tyBtnInShutterOpenCtrl.bValue			:= p_tyDO.bInShutterOpenCtrl;
		tyP0201OpsConv.tyIOMonitorXStd.tyBtnInShutterCloseCtrl.bValue			:= p_tyDO.bInShutterCloseCtrl;
		tyP0201OpsConv.tyIOMonitorXStd.tyBtnOutShutterOpenCtrl.bValue			:= p_tyDO.bOutShutterOpenCtrl;
		tyP0201OpsConv.tyIOMonitorXStd.tyBtnOutShutterCloseCtrl.bValue			:= p_tyDO.bOutShutterCloseCtrl;
		tyP0201OpsConv.tyIOMonitorXStd.tyBtnClamp1Ctrl.bValue					:= p_tyDO.bClamp1Ctrl;
		tyP0201OpsConv.tyIOMonitorXStd.tyBtnUnclamp1Ctrl.bValue					:= p_tyDO.bUnClamp1Ctrl;
		tyP0201OpsConv.tyIOMonitorXStd.tyBtnClamp2Ctrl.bValue					:= p_tyDO.bClamp2Ctrl;
		tyP0201OpsConv.tyIOMonitorXStd.tyBtnUnclamp2Ctrl.bValue					:= p_tyDO.bUnClamp2Ctrl;
		tyP0201OpsConv.tyIOMonitorXStd.tyBtnClamp3Ctrl.bValue					:= p_tyDO.bClamp3Ctrl;
		tyP0201OpsConv.tyIOMonitorXStd.tyBtnUnclamp3Ctrl.bValue					:= p_tyDO.bUnClamp3Ctrl;

	END_IF

	IF tyP0201OpsConv.tyIOMonitorXStdMachineSafety.tyLyr.uiRtStat.0 = FALSE THEN
		//Non Standard
		//Digital Input
		tyP0201OpsConv.tyIOMonitorXStdMachineSafety.tyBtnSafetyRlySig.bValue					:= p_tyDI.bSafetyRlySig;
		tyP0201OpsConv.tyIOMonitorXStdMachineSafety.tyBtnEStop.bValue						:= p_tyDI.bEStopSig;
		tyP0201OpsConv.tyIOMonitorXStdMachineSafety.tyBtnCoverSWSig.bValue					:= p_tyDI.bCoverSWSig;
		tyP0201OpsConv.tyIOMonitorXStdMachineSafety.tyBtnUBA.bValue							:= p_tyDI.bUBA;
		tyP0201OpsConv.tyIOMonitorXStdMachineSafety.tyBtnDSB.bValue							:= p_tyDI.bDSB;
		tyP0201OpsConv.tyIOMonitorXStdMachineSafety.tyBtnUBAStat.bValue						:= p_tyDI.bUBAStat;
		tyP0201OpsConv.tyIOMonitorXStdMachineSafety.tyBtnConvLftSen.bValue					:= p_tyDI.bConvLftSen;
		tyP0201OpsConv.tyIOMonitorXStdMachineSafety.tyBtnConvRgtSen.bValue					:= p_tyDI.bConvRgtSen;
		tyP0201OpsConv.tyIOMonitorXStdMachineSafety.tyBtnPressureSW.bValue					:= p_tyDI.bPressureSW;
		tyP0201OpsConv.tyIOMonitorXStdMachineSafety.tyBtnThermalPrtSig.bValue				:= p_tyDI.bThermalPrtSig;
		tyP0201OpsConv.tyIOMonitorXStdMachineSafety.tyBtnCoatingSen.bValue					:= p_tyDI.bCoatingSen;
		tyP0201OpsConv.tyIOMonitorXStdMachineSafety.tyBtnUSWidthChkSen.bValue				:= p_tyDI.bUSWidthChkSen;
		tyP0201OpsConv.tyIOMonitorXStdMachineSafety.tyBtnDSWidthChkSen.bValue				:= p_tyDI.bDSWidthChkSen;
		tyP0201OpsConv.tyIOMonitorXStdMachineSafety.tyBtnInvertHomeSen.bValue				:= p_tyDI.bInvertHomeSen;
		tyP0201OpsConv.tyIOMonitorXStdMachineSafety.tyBtnInvertRemoteSen.bValue				:= p_tyDI.bInvertRemoteSen;
		tyP0201OpsConv.tyIOMonitorXStdMachineSafety.tyBtnInletShutterOpenRS.bValue			:= p_tyDI.bInShutterOpenRS;
		tyP0201OpsConv.tyIOMonitorXStdMachineSafety.tyBtnInletShutterCloseRS.bValue			:= p_tyDI.bInShutterCloseRS;
		tyP0201OpsConv.tyIOMonitorXStdMachineSafety.tyBtnOutletShutterOpenRS.bValue			:= p_tyDI.bOutShutterOpenRS;
		tyP0201OpsConv.tyIOMonitorXStdMachineSafety.tyBtnOutletShutterCloseRS.bValue			:= p_tyDI.bOutShutterCloseRS;
		tyP0201OpsConv.tyIOMonitorXStdMachineSafety.tyBtnClamp2Sen.bValue					:= p_tyDI.bClamp2Sen;
		tyP0201OpsConv.tyIOMonitorXStdMachineSafety.tyBtnClamp3Sen.bValue					:= p_tyDI.bClamp3Sen;
		tyP0201OpsConv.tyIOMonitorXStdMachineSafety.tyBtnClampRS1.bValue						:= p_tyDI.bClampRS1;
		tyP0201OpsConv.tyIOMonitorXStdMachineSafety.tyBtnUnClampRS1.bValue					:= p_tyDI.bUnClampRS1;
		tyP0201OpsConv.tyIOMonitorXStdMachineSafety.tyBtnClampRS2.bValue						:= p_tyDI.bClampRS2;
		tyP0201OpsConv.tyIOMonitorXStdMachineSafety.tyBtnUnClampRS2.bValue					:= p_tyDI.bUnClampRS2;
		tyP0201OpsConv.tyIOMonitorXStdMachineSafety.tyBtnClampRS3.bValue						:= p_tyDI.bClampRS3;
		tyP0201OpsConv.tyIOMonitorXStdMachineSafety.tyBtnUnClampRS3.bValue					:= p_tyDI.bUnClampRS3;
		//ADD
		tyP0201OpsConv.tyIOMonitorXStdMachineSafety.tyBtnCoverSWSig2.bValue					:= p_tyDI.bCoverSWSig2;
		tyP0201OpsConv.tyIOMonitorXStdMachineSafety.tyBtnSafetySigFromUS.bValue				:= p_tyDI.bSafetySigFromUS;
		tyP0201OpsConv.tyIOMonitorXStdMachineSafety.tyBtnSafetySigFromDS.bValue				:= p_tyDI.bSafetySigFromDS;
		tyP0201OpsConv.tyIOMonitorXStdMachineSafety.tyBtnUnlockCoverSigFromUS.bValue		:= p_tyDI.bUnlockCoverSigFromUS;
		tyP0201OpsConv.tyIOMonitorXStdMachineSafety.tyBtnUnlockCoverSigFromDS.bValue		:= p_tyDI.bUnlockCoverSigFromDS;
		tyP0201OpsConv.tyIOMonitorXStdMachineSafety.tyBtnCoverUnlockPB1.bValue				:= p_tyDI.bCoverUnlockPB1;
		//Digital Output
		tyP0201OpsConv.tyIOMonitorXStdMachineSafety.tyBtnSafetyRlyRst.bValue					:= p_tyDO.bSafetyRlyRst;
		tyP0201OpsConv.tyIOMonitorXStdMachineSafety.tyBtnTLGreen.bValue						:= p_tyDO.bTLGreen;
		tyP0201OpsConv.tyIOMonitorXStdMachineSafety.tyBtnTLAmber.bValue						:= p_tyDO.bTLAmber;
		tyP0201OpsConv.tyIOMonitorXStdMachineSafety.tyBtnTLRed.bValue						:= p_tyDO.bTLRed;
		tyP0201OpsConv.tyIOMonitorXStdMachineSafety.tyBtnTLBlue.bValue						:= p_tyDO.bTLBlue;
		tyP0201OpsConv.tyIOMonitorXStdMachineSafety.tyBtnTLWhite.bValue						:= p_tyDO.bTLWhite;
		tyP0201OpsConv.tyIOMonitorXStdMachineSafety.tyBtnBuzzer.bValue						:= p_tyDO.bBuz;
		tyP0201OpsConv.tyIOMonitorXStdMachineSafety.tyBtnCoatingRetCtrl.bValue				:= p_tyDO.bCoatingStprRet;
		tyP0201OpsConv.tyIOMonitorXStdMachineSafety.tyBtnUSB.bValue							:= p_tyDO.bUSB;
		tyP0201OpsConv.tyIOMonitorXStdMachineSafety.tyBtnDBA.bValue							:= p_tyDO.bDBA;
		tyP0201OpsConv.tyIOMonitorXStdMachineSafety.tyBtnDBAStat.bValue						:= p_tyDO.bDBAStat;
		tyP0201OpsConv.tyIOMonitorXStdMachineSafety.tyBtnConvMtrCW.bValue					:= p_tyDO.bConvMtrCW;
		tyP0201OpsConv.tyIOMonitorXStdMachineSafety.tyBtnConvMtrCCW.bValue					:= p_tyDO.bConvMtrCCW;
		tyP0201OpsConv.tyIOMonitorXStdMachineSafety.tyBtnInvertHome.bValue					:= p_tyDO.bInvertHome;
		tyP0201OpsConv.tyIOMonitorXStdMachineSafety.tyBtnInvertRemote.bValue					:= p_tyDO.bInvertRemote;
		tyP0201OpsConv.tyIOMonitorXStdMachineSafety.tyBtnInvertBrake.bValue					:= p_tyDO.bInvertBrake;
		tyP0201OpsConv.tyIOMonitorXStdMachineSafety.tyBtnMtrPwrRly.bValue					:= p_tyDO.bMtrPwrRly;
		tyP0201OpsConv.tyIOMonitorXStdMachineSafety.tyBtnInShutterOpenCtrl.bValue			:= p_tyDO.bInShutterOpenCtrl;
		tyP0201OpsConv.tyIOMonitorXStdMachineSafety.tyBtnInShutterCloseCtrl.bValue			:= p_tyDO.bInShutterCloseCtrl;
		tyP0201OpsConv.tyIOMonitorXStdMachineSafety.tyBtnOutShutterOpenCtrl.bValue			:= p_tyDO.bOutShutterOpenCtrl;
		tyP0201OpsConv.tyIOMonitorXStdMachineSafety.tyBtnOutShutterCloseCtrl.bValue			:= p_tyDO.bOutShutterCloseCtrl;
		tyP0201OpsConv.tyIOMonitorXStdMachineSafety.tyBtnClamp1Ctrl.bValue					:= p_tyDO.bClamp1Ctrl;
		tyP0201OpsConv.tyIOMonitorXStdMachineSafety.tyBtnUnclamp1Ctrl.bValue					:= p_tyDO.bUnClamp1Ctrl;
		tyP0201OpsConv.tyIOMonitorXStdMachineSafety.tyBtnClamp2Ctrl.bValue					:= p_tyDO.bClamp2Ctrl;
		tyP0201OpsConv.tyIOMonitorXStdMachineSafety.tyBtnUnclamp2Ctrl.bValue					:= p_tyDO.bUnClamp2Ctrl;
		tyP0201OpsConv.tyIOMonitorXStdMachineSafety.tyBtnClamp3Ctrl.bValue					:= p_tyDO.bClamp3Ctrl;
		tyP0201OpsConv.tyIOMonitorXStdMachineSafety.tyBtnUnclamp3Ctrl.bValue					:= p_tyDO.bUnClamp3Ctrl;
		// ADD
		tyP0201OpsConv.tyIOMonitorXStdMachineSafety.tyBtnTopCvrUnlckToDS.bValue					:= p_tyDO.bTopCvrUnlckToDS;
		tyP0201OpsConv.tyIOMonitorXStdMachineSafety.tyBtnTopCvrUnlckToUS.bValue					:= p_tyDO.bTopCvrUnlckToUS;
		tyP0201OpsConv.tyIOMonitorXStdMachineSafety.tyBtniMachineSafetySigToDS.bValue			:= p_tyDO.bMachineSafetySigToDS;
		tyP0201OpsConv.tyIOMonitorXStdMachineSafety.tyBtnMachineSafetySigToUS.bValue			:= p_tyDO.bMachineSafetySigToUS;
		tyP0201OpsConv.tyIOMonitorXStdMachineSafety.tyBtnPBLED1.bValue							:= p_tyDO.bCoverPBLED1;
		tyP0201OpsConv.tyIOMonitorXStdMachineSafety.tyBtnBypassTopCover1.bValue					:= p_tyDO.bBypassTopCover1;
		tyP0201OpsConv.tyIOMonitorXStdMachineSafety.tyBtnSafetyTopCoverSWCoil1.bValue			:= p_tyDO.bSafetyTopCoverSWCoil1;

	END_IF

END_ACTION
```

#### Act_OptP0201ChgParam.st
```iecst
ACTION Act_OptP0201ChgParam:

	tyP0201OpsConv.tyOps.tyBtnChgParam.uiRtStat.0	:= NOT(p_tyMcParamCurr.bChgParamEn);

	//Control
	IF tyP0201OpsConv.tyOps.tyBtnChgParam.bRtCompl = TRUE THEN
		tyP0201OpsConv.tyOps.tyBtnChgParam.bRtCompl	:= FALSE;

		tyProdRcpCurrRcpWr	:= p_tyProdRcpCurrRcp0;

		tyP0201OpsConv.tyChgParam.tyDrpDnMcMode.usiValueIdx		:= p_tyProdRcpCurrRcp0.usiMcMod;
		tyP0201OpsConv.tyChgParam.tyDrpDnFlippedBrd.usiValueIdx	:= p_tyProdRcpCurrRcp0.usiFlippedBrd;
		tyP0201OpsConv.tyChgParam.tyNumProdWidth.diValue		:= p_tyProdRcpCurrRcp0.diWidthInUM;

		fUIInRtStatOff(ADR(tyP0201OpsConv.tyChgParam.tyLyr.uiRtStat));

	END_IF

	tyP0201OpsConv.tyOps.tyBtnChgParam.bValue	:= tyP0201OpsConv.tyChgParam.tyLyr.uiRtStat.0 = FALSE;

	IF tyP0201OpsConv.tyChgParam.tyLyr.uiRtStat.0 = FALSE THEN

		IF tyP0201OpsConv.tyChgParam.tyBtnSave.bRtCompl = TRUE THEN

			tyProdRcpCurrRcpWr.usiMcMod			:= tyP0201OpsConv.tyChgParam.tyDrpDnMcMode.usiValueIdx;
			tyProdRcpCurrRcpWr.usiFlippedBrd	:= tyP0201OpsConv.tyChgParam.tyDrpDnFlippedBrd.usiValueIdx;
			tyProdRcpCurrRcpWr.diWidthInUM		:= tyP0201OpsConv.tyChgParam.tyNumProdWidth.diValue;

			eProdRcpAct	:= ProdRcpActWriteCurrRcpParam;

			IF p_eProdRcpStatus = Done AND p_eProdRcpStat = ProdRcpActWriteCurrRcpParam THEN
				eProdRcpAct	:= ProdRcpActIdle;

				//UIP0400
				tyP0400ProdSel.tyProdSel.tyTxtMcMod.usiValueIdx			:= p_tyProdRcpCurrRcp0.usiMcMod;
				tyP0400ProdSel.tyProdSel.tyTxtFlippedBrd.usiValueIdx	:= p_tyProdRcpCurrRcp0.usiFlippedBrd;
				tyP0400ProdSel.tyProdSel.tyNumProdWidth.diValue			:= p_tyProdRcpCurrRcp0.diWidthInUM;

				tyP0201OpsConv.tyChgParam.tyBtnSave.bRtCompl	:= FALSE;
				tyP0201OpsConv.tyChgParam.tyBtnSave.bValue		:= FALSE;

				fUIInRtStatHide(ADR(tyP0201OpsConv.tyChgParam.tyLyr.uiRtStat));

			ELSIF p_eProdRcpStatus = Error THEN
				p_tyC0008MsgBox ACCESS ADR(tyP0201OpsConv.tyMsgBoxSaveErr);

				IF tyP0201OpsConv.tyMsgBoxSaveErr.tyBtnNo.bRtCompl = TRUE THEN
					tyP0201OpsConv.tyMsgBoxSaveErr.tyBtnNo.bRtCompl	:= FALSE;
					tyP0201OpsConv.tyMsgBoxSaveErr.tyBtnNo.bValue	:= FALSE;

					p_tyC0008MsgBox ACCESS ADR(tyP0201OpsConv.tyMsgBoxHide);

					//Restore Param
					tyProdRcpCurrRcpWr	:= p_tyProdRcpCurrRcp0;

					tyP0201OpsConv.tyChgParam.tyBtnSave.bRtCompl	:= FALSE;
					tyP0201OpsConv.tyChgParam.tyBtnSave.bValue	:= FALSE;

					fUIInRtStatHide(ADR(tyP0201OpsConv.tyChgParam.tyLyr.uiRtStat));

				END_IF

			END_IF

		ELSIF tyP0201OpsConv.tyChgParam.tyBtnCancel.bRtCompl = TRUE THEN
			tyP0201OpsConv.tyChgParam.tyBtnCancel.bRtCompl	:= FALSE;
			tyP0201OpsConv.tyChgParam.tyBtnCancel.bValue		:= FALSE;

			fUIInRtStatHide(ADR(tyP0201OpsConv.tyChgParam.tyLyr.uiRtStat));
		END_IF

	END_IF

	//Mask
	tyP0201OpsConv.tyOps.tyBtnChgParam.uiMaskRtStat.0	:= p_tyUsrMgmtCurrAccessRgt.bChgParam AND p_bOpsStatusStop;

END_ACTION
```

#### Act_OptP0201AccDat.st
```iecst
ACTION Act_OptP0201AccDat:

	IF g_tyP0200Opt.tyOpt.tyBtnAccDat.bRtCompl = TRUE THEN
		g_tyP0200Opt.tyOpt.tyBtnAccDat.bRtCompl	:= FALSE;
		tyAccData.bAccDatStart					:= TRUE;
	END_IF

	//Button Appearance
	IF tyAccData.bAccDatReq = TRUE THEN
		IF tyAccData.bAccDatStart = FALSE THEN
			fbAccDatBlinkTm(IN := TRUE);

			IF fbAccDatBlinkTm.Q THEN
				fbAccDatBlinkTm(IN := FALSE);

				IF g_tyP0200Opt.tyOpt.tyBitmapAccDat.usiValueIdx = 1 THEN
					g_tyP0200Opt.tyOpt.tyBitmapAccDat.usiValueIdx	:= 0;
				ELSE
					g_tyP0200Opt.tyOpt.tyBitmapAccDat.usiValueIdx	:= 1;
				END_IF
			END_IF
		ELSE
			fbAccDatBlinkTm(IN := FALSE);
			g_tyP0200Opt.tyOpt.tyBitmapAccDat.usiValueIdx			:= 1;
		END_IF

	ELSE
		fbAccDatBlinkTm(IN := FALSE);
		g_tyP0200Opt.tyOpt.tyBitmapAccDat.usiValueIdx				:= 0;
	END_IF

	//Mask
	IF tyMcParamData.tyRcpMcParam.tyUpstream.eComm = McSetCommModSMEMA THEN
		IF tyAccData.bAccDatAllow AND tyAccData.bAccDatReq AND NOT tyFollowerData.bAutoAccDatOut AND tyAccData.bAccDatStart = FALSE THEN
			fUIInRtStatHide(ADR(g_tyP0200Opt.tyOpt.tyBtnAccDat.uiMaskRtStat));
		ELSE
			fUIInRtStatOff(ADR(g_tyP0200Opt.tyOpt.tyBtnAccDat.uiMaskRtStat));
		END_IF
	ELSIF tyMcParamData.tyRcpMcParam.tyUpstream.eComm = McSetCommModHermes THEN
		IF tyAccData.bAccDatAllow AND tyAccData.bAccDatReq AND tyAccData.bAccDatStart = FALSE THEN
			fUIInRtStatHide(ADR(g_tyP0200Opt.tyOpt.tyBtnAccDat.uiMaskRtStat));
		ELSE
			fUIInRtStatOff(ADR(g_tyP0200Opt.tyOpt.tyBtnAccDat.uiMaskRtStat));
		END_IF
	END_IF

END_ACTION
```

#### Act_OptP0201Keypad.st
```iecst
ACTION Act_OptP0201Keypad:

	IF fUIOutRtStatTPIsOpen(ADR(tyP0201OpsConv.tyChgParam.tyNumProdWidth.uiRtStat)) THEN
		tyProperty.tyKeypad.tyTxtTitle.sTxt	:= tyP0201OpsConv.tyChgParam.tyNumProdWidth.sKeypadTitle;

	END_IF

END_ACTION
```
